(** AXIS Z **)
	(* Brake timer *)
		tonZBrake(PT:=T#20S);
		IF GV_Axes.stAxisZ.bPowerEnable AND GV_Axes.stAxisZ.stDriveAx8206.AxisRef.Status.NotMoving THEN
			tonZBrake.IN:=TRUE;
		ELSE
			tonZBrake.IN:=FALSE;
		END_IF
	(* Setup *)
		GV_Axes.stAxisZ.bPresence:=TRUE; // Axis Presence
		fbEventGroupAssignement(iEventGroup:=GV_Axes.stAxisZ.iEventGroup);
		GV_Axes.stAxisZ.strIdHMI:='Z'; // String for events on HMI
		GV_Axes.stAxisZ.iIdHMI:=UDINT_TO_INT(GV_Axes.stAxisZ.stDriveAx8206.AxisRef.NcToPlc.AxisId); // Number for events on HMI
		(*Power*)
			IF ((GV_OpMode.eOpMode=ENUM_OpMode.INIT AND (GV_Axes.stAxisZ.bAutoCmdAbs OR (GV_Axes.stAxisZ.bPowerEnable AND (NOT tonZBrake.Q)))) // INIT
			OR (GV_OpMode.eOpMode=ENUM_OpMode.AUTO AND (GV_Axes.stAxisZ.bAutoCmdAbs OR (GV_Axes.stAxisZ.bPowerEnable AND (NOT tonZBrake.Q)))) // AUTO
			OR (GV_OpMode.eOpMode=ENUM_OpMode.MANU AND (((NOT GV_Handwheel.aId[1].bEnable) AND (GV_Axes.eJogAxisRequest=ENUM_Axis_Select.Z OR GV_Axes.eJogAxisSelect=ENUM_Axis_Select.Z)) OR (GV_Handwheel.aId[1].bEnable AND GV_Handwheel.aId[1].eAxisSelect=ENUM_Axis_Select.Z)))) // MANU
			AND ((GV_General.bSafety AND GV_General.bPower AND (NOT GV_Axes.stAxisZ.bAlAxisFault)) OR (GV_Axes.stAxisZ.bPowerEnable AND ((GV_Axes.stAxisZ.bStopExecute AND (NOT GV_Axes.stAxisZ.bStopDone))) OR (GV_Axes.stAxisZ.bHaltExecute AND (NOT GV_Axes.stAxisZ.bHaltDone)))) AND (NOT GV_General.bRebootRequest) AND (NOT GV_General.bShutdownRequest) THEN
				GV_Axes.stAxisZ.bPowerEnable:=TRUE;
			ELSE
				GV_Axes.stAxisZ.bPowerEnable:=FALSE;
			END_IF
		(*Stop*)
			GV_Axes.stAxisZ.bStopExecute:=(NOT GV_General.bSafety) OR (NOT GV_General.bPower) OR GV_General.bRebootRequest OR GV_General.bShutdownRequest (*OR (GV_OpMode.eOpMode=ENUM_OpMode.AUTO AND GV_Cycle.bCycleInProgress AND (NOT GV_Cycle.bStartStop))*); // Have to stop
		(*Halt*)
			GV_Axes.stAxisZ.bHaltExecute:=(GV_OpMode.eOpMode=ENUM_OpMode.AUTO AND GV_Cycle.bCycleInProgress AND (NOT GV_Cycle.bStartStop)); // Have to halt
		(*Abort*)
			//GV_Axes.stAxisZ.bAbort:=(NOT GV_Axes.stAxisZ.stDriveAx8206.AxisRef.Status.NotMoving) AND (GV_OpMode.eOpMode=ENUM_OpMode.AUTO AND GV_Cycle.bCycleInProgress AND (NOT GV_Cycle.bStartStop)); // Have to abort
		(*Reset*)
			GV_Axes.stAxisZ.bEventAck:=GV_HMI.bEventAck; // Events Acknowledgement	
		(*Jog*)
			GV_Axes.stAxisZ.bJogEnable:=GV_OpMode.eOpMode=ENUM_OpMode.MANU AND GV_Axes.stAxisZ.stDriveAx8206.AxisRef.Status.Operational AND (NOT GV_Axes.stAxisZ.bAlAxisFault) AND
			((GV_Handwheel.aId[1].bEnable AND GV_Handwheel.aId[1].eAxisSelect=ENUM_Axis_Select.Z) OR ((NOT GV_Handwheel.aId[1].bEnable) AND GV_HMI.iCurrentScreenNumber=210 AND GV_Axes.eJogAxisSelect=ENUM_Axis_Select.Z));
			IF GV_Axes.stAxisZ.bJogEnable AND (NOT GV_Handwheel.aId[1].bEnable) THEN // Jog from HMI
				GV_Axes.stAxisZ.eJogMode:=TC2_MC2.E_JogMode.MC_JOGMODE_CONTINOUS; // Jog Mode
				GV_Axes.stAxisZ.bJogPlus:=GV_HMI.stAxes.bButtonPlus; // Jog +
				GV_Axes.stAxisZ.bJogMinus:=GV_HMI.stAxes.bButtonMinus; // Jog -
				GV_Axes.stAxisZ.lrJogPos:=0; // Jog Position -> Only in mode INCHING
				GV_Axes.stAxisZ.lrJogVel:=GV_Axes.lrVelocityAxisZ; // Jog Velocity
				GV_Axes.stAxisZ.lrJogAcc:=0; // Jog Acceleration -> see the Axis Configuration in the System Manager
				GV_Axes.stAxisZ.lrJogDec:=0; // Jog Decelration -> see the Axis Configuration in the System Manager
				GV_Axes.stAxisZ.lrJogJerk:=0; // Jog Jerk -> see the Axis Configuration in the System Manager
			ELSIF GV_Axes.stAxisZ.bJogEnable AND GV_Handwheel.aId[1].bEnable AND GV_Handwheel.aId[1].bJogRequestRisingEdge THEN // Jog from Handwheel
				GV_Axes.stAxisZ.eJogMode:=TC2_MC2.E_JogMode.MC_JOGMODE_INCHING; // Jog Mode
				GV_Axes.stAxisZ.bJogPlus:=(GV_Handwheel.aId[1].eJogDirection=ENUM_Jog_Direction.Plus); // Jog +
				GV_Axes.stAxisZ.bJogMinus:=(GV_Handwheel.aId[1].eJogDirection=ENUM_Jog_Direction.Minus); // Jog -
				GV_Axes.stAxisZ.lrJogPos:=GV_Handwheel.aId[1].lrJogIncrRequest; // Jog Position
				GV_Axes.stAxisZ.lrJogVel:=GV_Axes.lrJogMaxSpeedAxisZ;//GV_Axes.lrVelocityAxisZ; // Jog Velocity
				GV_Axes.stAxisZ.lrJogAcc:=0; // Jog Acceleration -> see the Axis Configuration in the System Manager
				GV_Axes.stAxisZ.lrJogDec:=0; // Jog Decelration -> see the Axis Configuration in the System Manager
				GV_Axes.stAxisZ.lrJogJerk:=0; // Jog Jerk -> see the Axis Configuration in the System Manager
			ELSE
				GV_Axes.stAxisZ.bJogPlus:=FALSE; // Jog +
				GV_Axes.stAxisZ.bJogMinus:=FALSE; // Jog -
				GV_Axes.stAxisZ.lrJogPos:=0; // Jog Position
				GV_Axes.stAxisZ.lrJogVel:=0; // Jog Velocity
				GV_Axes.stAxisZ.lrJogAcc:=0; // Jog Acceleration -> see the Axis Configuration in the System Manager
				GV_Axes.stAxisZ.lrJogDec:=0; // Jog Decelration -> see the Axis Configuration in the System Manager
				GV_Axes.stAxisZ.lrJogJerk:=0; // Jog Jerk -> see the Axis Configuration in the System Manager				
			END_IF
		(*AUTO*)
			GV_Axes.stAxisZ.bAutoEnable:=GV_OpMode.eOpMode=ENUM_OpMode.AUTO AND GV_Cycle.bStartStop AND GV_Axes.stAxisZ.stDriveAx8206.AxisRef.Status.Operational AND (NOT GV_Axes.stAxisZ.bAlAxisFault);
			IF  GV_Axes.stAxisZ.bAutoEnable THEN
				GV_Axes.stAxisZ.lrAutoVelAbs:=GV_Axes.lrVelocityAxisZ; // AUTO Velocity
				GV_Axes.stAxisZ.lrAutoAccAbs:=0; // AUTO Acceleration -> see the Axis Configuration in the System Manager
				GV_Axes.stAxisZ.lrAutoDecAbs:=0; // AUTO Decelration -> see the Axis Configuration in the System Manager
				GV_Axes.stAxisZ.lrAutoJerkAbs:=0; // AUTO Jerk -> see the Axis Configuration in the System Manager
			ELSE
				GV_Axes.stAxisZ.lrAutoVelAbs:=0; // AUTO Velocity
				GV_Axes.stAxisZ.lrAutoAccAbs:=0; // AUTO Acceleration -> see the Axis Configuration in the System Manager
				GV_Axes.stAxisZ.lrAutoDecAbs:=0; // AUTO Decelration -> see the Axis Configuration in the System Manager
				GV_Axes.stAxisZ.lrAutoJerkAbs:=0; // AUTO Jerk -> see the Axis Configuration in the System Manager
			END_IF
		(*Referencing*)
			GV_Axes.stAxisZ.bSetOffsetExecute:=GV_OpMode.eOpMode=ENUM_OpMode.MANU AND GV_Axes.stAxisZ.stDriveAx8206.AxisRef.Status.Operational AND (NOT GV_Axes.stAxisZ.bAlAxisFault) AND GV_HMI.iCurrentScreenNumber=308 AND GV_Axes.eRefAxisSelect=ENUM_Axis_Select.Z AND GV_HMI.stAxes.rtButtonReferencingAxis.Q;
			GV_Axes.stAxisZ.bDeleteOffsetExecute:=FALSE; // Not used in the HMI, we can use it from here or add it in the HMI later if it's necessary	
		(*ReadParameter BOOL*)
			GV_Axes.stAxisZ.bReadbEnable:=(GV_Axes.stAxisZ.mcAxisReadParameterb=MC_AxisParameter.AxisEnMinSoftPosLimit OR GV_Axes.stAxisZ.mcAxisReadParameterb=MC_AxisParameter.AxisEnMaxSoftPosLimit) AND GV_Axes.stAxisZ.stDriveAx8206.AxisRef.Status.Operational;
			IF GV_Axes.stAxisZ.stDriveAx8206.AxisRef.Status.Operational THEN
				IF GV_Axes.stAxisZ.mcAxisReadParameterb=MC_AxisParameter.AxisEnMaxSoftPosLimit THEN
					IF GV_General.bIsBlinking05s THEN
						GV_Axes.stAxisZ.mcAxisReadParameterb:=MC_AxisParameter.AxisEnMinSoftPosLimit;
					ELSE
						IF GV_Axes.stAxisZ.bReadbValid THEN
							GV_Axes.stAxisZ.bReadEnMaxSoftPosLimit:=GV_Axes.stAxisZ.bReadbValue;
						END_IF
					END_IF
				ELSIF GV_Axes.stAxisZ.mcAxisReadParameterb=MC_AxisParameter.AxisEnMinSoftPosLimit THEN
					IF GV_General.bIsBlinking05s THEN
						GV_Axes.stAxisZ.mcAxisReadParameterb:=MC_AxisParameter.AxisEnMaxSoftPosLimit;
					ELSE
						IF GV_Axes.stAxisZ.bReadbValid THEN
							GV_Axes.stAxisZ.bReadEnMinSoftPosLimit:=GV_Axes.stAxisZ.bReadbValue;
						END_IF
					END_IF
				ELSE
					GV_Axes.stAxisZ.mcAxisReadParameterb:=MC_AxisParameter.AxisEnMinSoftPosLimit;
				END_IF
			END_IF
		(*ReadParameter LREAL*)
			GV_Axes.stAxisZ.bReadlrEnable:=(GV_Axes.stAxisZ.mcAxisReadParameterlr=MC_AxisParameter.AxisMinSoftPosLimit OR GV_Axes.stAxisZ.mcAxisReadParameterlr=MC_AxisParameter.AxisMaxSoftPosLimit) AND GV_Axes.stAxisZ.stDriveAx8206.AxisRef.Status.Operational;
			IF GV_Axes.stAxisZ.stDriveAx8206.AxisRef.Status.Operational THEN
				IF GV_Axes.stAxisZ.mcAxisReadParameterlr=MC_AxisParameter.AxisMaxSoftPosLimit THEN
					IF GV_General.bIsBlinking05s THEN
						GV_Axes.stAxisZ.mcAxisReadParameterlr:=MC_AxisParameter.AxisMinSoftPosLimit;
					ELSE
						IF GV_Axes.stAxisZ.bReadlrValid THEN
							GV_Axes.stAxisZ.lrReadMaxSoftPosLimit:=GV_Axes.stAxisZ.lrReadlrValue;
						END_IF
					END_IF
				ELSIF GV_Axes.stAxisZ.mcAxisReadParameterlr=MC_AxisParameter.AxisMinSoftPosLimit THEN
					IF (NOT GV_General.bIsBlinking05s) THEN
						GV_Axes.stAxisZ.mcAxisReadParameterlr:=MC_AxisParameter.AxisMaxSoftPosLimit;
					ELSE
						IF GV_Axes.stAxisZ.bReadlrValid THEN
							GV_Axes.stAxisZ.lrReadMinSoftPosLimit:=GV_Axes.stAxisZ.lrReadlrValue;
						END_IF
					END_IF
				ELSE
					GV_Axes.stAxisZ.mcAxisReadParameterlr:=MC_AxisParameter.AxisMinSoftPosLimit;
				END_IF
			END_IF	
		(*WriteParameter BOOL*)
// 			GV_Axes.stAxisZ.bWritebExecute:=GV_Axes.eRefAxisSelect=ENUM_Axis_Select.Z AND (GV_HMI.stAxes.rtButtonMinSofltLimit.Q OR GV_HMI.stAxes.rtButtonMaxSofltLimit.Q) AND GV_Axes.stAxisZ.stDriveAx8206.AxisRef.Status.Operational;
// 			IF GV_Axes.stAxisZ.stDriveAx8206.AxisRef.Status.Operational AND (NOT GV_Axes.stAxisZ.stDriveAx8206.AxisRef.Status.Moving) THEN
// 				IF GV_HMI.stAxes.rtButtonMinSofltLimit.Q THEN
// 					GV_Axes.stAxisZ.mcAxisWriteParameterb:=MC_AxisParameter.AxisEnMinSoftPosLimit;
// 					IF GV_Axes.stAxisZ.bReadEnMinSoftPosLimit THEN
// 						GV_Axes.stAxisZ.bWritebValue:=FALSE;
// 					ELSE
// 						GV_Axes.stAxisZ.bWritebValue:=TRUE;
// 					END_IF
// 				ELSIF GV_HMI.stAxes.rtButtonMaxSofltLimit.Q THEN
// 					GV_Axes.stAxisZ.mcAxisWriteParameterb:=MC_AxisParameter.AxisEnMaxSoftPosLimit;
// 					IF GV_Axes.stAxisZ.bReadEnMaxSoftPosLimit THEN
// 						GV_Axes.stAxisZ.bWritebValue:=FALSE;
// 					ELSE
// 						GV_Axes.stAxisZ.bWritebValue:=TRUE;
// 					END_IF
// 				END_IF
// 			END_IF
		(*WriteParameter LREAL*)
// 			bAxisZWrite1:=FALSE;
// 			bAxisZWrite2:=FALSE;
// 			bAxisZWrite3:=FALSE;
// 			bAxisZWrite4:=FALSE;
// 			IF GV_Tool_Magazine.stManipulator.ePositionMag=ENUM_Position_Magazine.Top THEN
// 				IF GV_Tool_Magazine.stManipulator.lrZPosition<>GV_Tool_Magazine.stManipulator.lrZTunnel THEN
// 					GV_Axes.stAxisZ.lrValueMax:=-10;
// 					GV_Axes.stAxisZ.lrValueMin:=-350;
// 					bAxisZWrite1:=TRUE;
// 				ELSE
// 					GV_Axes.stAxisZ.lrValueMax:=-10;
// 					GV_Axes.stAxisZ.lrValueMin:=-800;
// 					bAxisZWrite2:=TRUE;
// 				END_IF
// 			END_IF
// 			IF GV_Tool_Magazine.stManipulator.ePositionMag=ENUM_Position_Magazine.Bottom THEN
// 				IF GV_Tool_Magazine.stManipulator.lrZPosition<>GV_Tool_Magazine.stManipulator.lrZTunnel THEN
// 					GV_Axes.stAxisZ.lrValueMax:=-450;
// 					GV_Axes.stAxisZ.lrValueMin:=-800;
// 					bAxisZWrite3:=TRUE;
// 				ELSE
// 					GV_Axes.stAxisZ.lrValueMax:=-10;
// 					GV_Axes.stAxisZ.lrValueMin:=-800;
// 					bAxisZWrite4:=TRUE;
// 				END_IF
// 			END_IF
// 			rtAxisZWrite1(CLK:=bAxisZWrite1);
// 			rtAxisZWrite2(CLK:=bAxisZWrite2);
// 			rtAxisZWrite3(CLK:=bAxisZWrite3);
// 			rtAxisZWrite4(CLK:=bAxisZWrite4);
// 			IF rtAxisZWrite1.Q OR rtAxisZWrite2.Q OR rtAxisZWrite3.Q OR rtAxisZWrite4.Q THEN
// 				GV_Axes.stAxisZ.mcAxisWriteParameterlr:=MC_AxisParameter.AxisMaxSoftPosLimit;
// 				GV_Axes.stAxisZ.lrWritelrValue:=GV_Axes.stAxisZ.lrValueMax;
// 				bAxisZWriteMin:=FALSE;
// 				bAxisZWriteMax:=TRUE;
// 			END_IF
// 			IF bAxisZWriteMax AND GV_Axes.stAxisZ.bWritelrBusy THEN
// 				GV_Axes.stAxisZ.mcAxisWriteParameterlr:=MC_AxisParameter.AxisMinSoftPosLimit;
// 				GV_Axes.stAxisZ.lrWritelrValue:=GV_Axes.stAxisZ.lrValueMin;
// 				bAxisZWriteMin:=TRUE;
// 				bAxisZWriteMax:=FALSE;
// 			END_IF
// 			IF bAxisZWriteMin AND GV_Axes.stAxisZ.bWritelrBusy THEN
// 				bAxisZWriteMin:=FALSE;
// 				bAxisZWriteMax:=FALSE;
// 			END_IF
// 			GV_Axes.stAxisZ.bWritelrExecute:=(bAxisZWriteMax OR bAxisZWriteMin) AND GV_Axes.stAxisZ.bWritelrDone AND (NOT GV_Axes.stAxisZ.bWritelrBusy) AND GV_Axes.stAxisZ.stDriveAx8206.AxisRef.Status.Operational;
// 			
	(* Fb *)
		IF GV_Axes.stAxisZ.bPresence THEN
			fbAxisZ(
					stAxis:=GV_Axes.stAxisZ,
					);
		END_IF

(** AXIS Arm **)
	(* Setup *)
		GV_Axes.stAxisArm.bPresence:=TRUE; // Axis Presence
		fbEventGroupAssignement(iEventGroup:=GV_Axes.stAxisArm.iEventGroup);
		GV_Axes.stAxisArm.strIdHMI:='Arm'; // String for events on HMI
		GV_Axes.stAxisArm.iIdHMI:=UDINT_TO_INT(GV_Axes.stAxisArm.stDriveAx8206.AxisRef.NcToPlc.AxisId); // Number for events on HMI
		(*Power*)
			IF ((GV_General.bSafety AND GV_General.bPower AND (NOT GV_Axes.stAxisArm.bAlAxisFault)) OR (GV_Axes.stAxisArm.bPowerEnable AND ((GV_Axes.stAxisArm.bStopExecute AND (NOT GV_Axes.stAxisArm.bStopDone))) OR ((GV_Axes.stAxisArm.bHaltExecute AND (NOT GV_Axes.stAxisArm.bHaltDone))))) AND (NOT GV_General.bRebootRequest) AND (NOT GV_General.bShutdownRequest) THEN
				GV_Axes.stAxisArm.bPowerEnable:=TRUE;
			ELSE
				GV_Axes.stAxisArm.bPowerEnable:=FALSE;
			END_IF
		(*Stop*)
			GV_Axes.stAxisArm.bStopExecute:=(NOT GV_General.bSafety) OR (NOT GV_General.bPower) OR GV_General.bRebootRequest OR GV_General.bShutdownRequest (*OR (GV_OpMode.eOpMode=ENUM_OpMode.AUTO AND GV_Cycle.bCycleInProgress AND (NOT GV_Cycle.bStartStop))*); // Have to stop
		(*Halt*)
			GV_Axes.stAxisArm.bHaltExecute:=(GV_OpMode.eOpMode=ENUM_OpMode.AUTO AND GV_Cycle.bCycleInProgress AND (NOT GV_Cycle.bStartStop)); // Have to halt
		(*Abort*)
			//GV_Axes.stAxisArm.bAbort:=(NOT GV_Axes.stAxisArm.stDriveAx8206.AxisRef.Status.NotMoving) AND (GV_OpMode.eOpMode=ENUM_OpMode.AUTO AND GV_Cycle.bCycleInProgress AND (NOT GV_Cycle.bStartStop)); // Have to abort
		(*Reset*)
			GV_Axes.stAxisArm.bEventAck:=GV_HMI.bEventAck; // Events Acknowledgement	
		(*Jog*)
			GV_Axes.stAxisArm.bJogEnable:=GV_OpMode.eOpMode=ENUM_OpMode.MANU AND GV_Axes.stAxisArm.stDriveAx8206.AxisRef.Status.Operational AND (NOT GV_Axes.stAxisArm.bAlAxisFault) AND
			((GV_Handwheel.aId[1].bEnable AND GV_Handwheel.aId[1].eAxisSelect=ENUM_Axis_Select.Arm) OR ((NOT GV_Handwheel.aId[1].bEnable) AND GV_HMI.iCurrentScreenNumber=210 AND GV_Axes.eJogAxisSelect=ENUM_Axis_Select.Arm));
			IF GV_Axes.stAxisArm.bJogEnable AND (NOT GV_Handwheel.aId[1].bEnable) THEN // Jog from HMI
				GV_Axes.stAxisArm.eJogMode:=TC2_MC2.E_JogMode.MC_JOGMODE_CONTINOUS; // Jog Mode
				GV_Axes.stAxisArm.bJogPlus:=GV_HMI.stAxes.bButtonPlus; // Jog +
				GV_Axes.stAxisArm.bJogMinus:=GV_HMI.stAxes.bButtonMinus; // Jog -
				GV_Axes.stAxisArm.lrJogPos:=0; // Jog Position -> Only in mode INCHING
				GV_Axes.stAxisArm.lrJogVel:=GV_Axes.lrVelocityAxisArm; // Jog Velocity
				GV_Axes.stAxisArm.lrJogAcc:=0; // Jog Acceleration -> see the Axis Configuration in the System Manager
				GV_Axes.stAxisArm.lrJogDec:=0; // Jog Decelration -> see the Axis Configuration in the System Manager
				GV_Axes.stAxisArm.lrJogJerk:=0; // Jog Jerk -> see the Axis Configuration in the System Manager
			ELSIF GV_Axes.stAxisArm.bJogEnable AND GV_Handwheel.aId[1].bEnable AND GV_Handwheel.aId[1].bJogRequestRisingEdge THEN // Jog from Handwheel
				GV_Axes.stAxisArm.eJogMode:=TC2_MC2.E_JogMode.MC_JOGMODE_INCHING; // Jog Mode
				GV_Axes.stAxisArm.bJogPlus:=(GV_Handwheel.aId[1].eJogDirection=ENUM_Jog_Direction.Plus); // Jog +
				GV_Axes.stAxisArm.bJogMinus:=(GV_Handwheel.aId[1].eJogDirection=ENUM_Jog_Direction.Minus); // Jog -
				GV_Axes.stAxisArm.lrJogPos:=GV_Handwheel.aId[1].lrJogIncrRequest; // Jog Position
				GV_Axes.stAxisArm.lrJogVel:=GV_Axes.lrJogMaxSpeedAxisArm;//GV_Axes.lrVelocityAxisArm; // Jog Velocity
				GV_Axes.stAxisArm.lrJogAcc:=0; // Jog Acceleration -> see the Axis Configuration in the System Manager
				GV_Axes.stAxisArm.lrJogDec:=0; // Jog Decelration -> see the Axis Configuration in the System Manager
				GV_Axes.stAxisArm.lrJogJerk:=0; // Jog Jerk -> see the Axis Configuration in the System Manager
			ELSE
				GV_Axes.stAxisArm.bJogPlus:=FALSE; // Jog +
				GV_Axes.stAxisArm.bJogMinus:=FALSE; // Jog -
				GV_Axes.stAxisArm.lrJogPos:=0; // Jog Position
				GV_Axes.stAxisArm.lrJogVel:=0; // Jog Velocity
				GV_Axes.stAxisArm.lrJogAcc:=0; // Jog Acceleration -> see the Axis Configuration in the System Manager
				GV_Axes.stAxisArm.lrJogDec:=0; // Jog Decelration -> see the Axis Configuration in the System Manager
				GV_Axes.stAxisArm.lrJogJerk:=0; // Jog Jerk -> see the Axis Configuration in the System Manager				
			END_IF
		(*AUTO*)
			GV_Axes.stAxisArm.bAutoEnable:=GV_OpMode.eOpMode=ENUM_OpMode.AUTO AND GV_Cycle.bStartStop AND GV_Axes.stAxisArm.stDriveAx8206.AxisRef.Status.Operational AND (NOT GV_Axes.stAxisArm.bAlAxisFault);
			IF  GV_Axes.stAxisArm.bAutoEnable THEN
				GV_Axes.stAxisArm.lrAutoVelAbs:=GV_Axes.lrVelocityAxisArm; // AUTO Velocity
				GV_Axes.stAxisArm.lrAutoAccAbs:=0; // AUTO Acceleration -> see the Axis Configuration in the System Manager
				GV_Axes.stAxisArm.lrAutoDecAbs:=0; // AUTO Decelration -> see the Axis Configuration in the System Manager
				GV_Axes.stAxisArm.lrAutoJerkAbs:=0; // AUTO Jerk -> see the Axis Configuration in the System Manager
			ELSE
				GV_Axes.stAxisArm.lrAutoVelAbs:=0; // AUTO Velocity
				GV_Axes.stAxisArm.lrAutoAccAbs:=0; // AUTO Acceleration -> see the Axis Configuration in the System Manager
				GV_Axes.stAxisArm.lrAutoDecAbs:=0; // AUTO Decelration -> see the Axis Configuration in the System Manager
				GV_Axes.stAxisArm.lrAutoJerkAbs:=0; // AUTO Jerk -> see the Axis Configuration in the System Manager
			END_IF
		(*Referencing*)
			GV_Axes.stAxisArm.bSetOffsetExecute:=GV_OpMode.eOpMode=ENUM_OpMode.MANU AND GV_Axes.stAxisArm.stDriveAx8206.AxisRef.Status.Operational AND (NOT GV_Axes.stAxisArm.bAlAxisFault) AND GV_HMI.iCurrentScreenNumber=308 AND GV_Axes.eRefAxisSelect=ENUM_Axis_Select.Arm AND GV_HMI.stAxes.rtButtonReferencingAxis.Q;
			GV_Axes.stAxisArm.bDeleteOffsetExecute:=FALSE; // Not used in the HMI, we can use it from here or add it in the HMI later if it's necessary	
		(*ReadParameter BOOL*)
			GV_Axes.stAxisArm.bReadbEnable:=(GV_Axes.stAxisArm.mcAxisReadParameterb=MC_AxisParameter.AxisEnMinSoftPosLimit OR GV_Axes.stAxisArm.mcAxisReadParameterb=MC_AxisParameter.AxisEnMaxSoftPosLimit) AND GV_Axes.stAxisArm.stDriveAx8206.AxisRef.Status.Operational;
			IF GV_Axes.stAxisArm.stDriveAx8206.AxisRef.Status.Operational THEN
				IF GV_Axes.stAxisArm.mcAxisReadParameterb=MC_AxisParameter.AxisEnMaxSoftPosLimit THEN
					IF GV_General.bIsBlinking05s THEN
						GV_Axes.stAxisArm.mcAxisReadParameterb:=MC_AxisParameter.AxisEnMinSoftPosLimit;
					ELSE
						IF GV_Axes.stAxisArm.bReadbValid THEN
							GV_Axes.stAxisArm.bReadEnMaxSoftPosLimit:=GV_Axes.stAxisArm.bReadbValue;
						END_IF
					END_IF
				ELSIF GV_Axes.stAxisArm.mcAxisReadParameterb=MC_AxisParameter.AxisEnMinSoftPosLimit THEN
					IF GV_General.bIsBlinking05s THEN
						GV_Axes.stAxisArm.mcAxisReadParameterb:=MC_AxisParameter.AxisEnMaxSoftPosLimit;
					ELSE
						IF GV_Axes.stAxisArm.bReadbValid THEN
							GV_Axes.stAxisArm.bReadEnMinSoftPosLimit:=GV_Axes.stAxisArm.bReadbValue;
						END_IF
					END_IF
				ELSE
					GV_Axes.stAxisArm.mcAxisReadParameterb:=MC_AxisParameter.AxisEnMinSoftPosLimit;
				END_IF
			END_IF
		(*ReadParameter LREAL*)
			GV_Axes.stAxisArm.bReadlrEnable:=(GV_Axes.stAxisArm.mcAxisReadParameterlr=MC_AxisParameter.AxisMinSoftPosLimit OR GV_Axes.stAxisArm.mcAxisReadParameterlr=MC_AxisParameter.AxisMaxSoftPosLimit) AND GV_Axes.stAxisArm.stDriveAx8206.AxisRef.Status.Operational;
			IF GV_Axes.stAxisArm.stDriveAx8206.AxisRef.Status.Operational THEN
				IF GV_Axes.stAxisArm.mcAxisReadParameterlr=MC_AxisParameter.AxisMaxSoftPosLimit THEN
					IF GV_General.bIsBlinking05s THEN
						GV_Axes.stAxisArm.mcAxisReadParameterlr:=MC_AxisParameter.AxisMinSoftPosLimit;
					ELSE
						IF GV_Axes.stAxisArm.bReadlrValid THEN
							GV_Axes.stAxisArm.lrReadMaxSoftPosLimit:=GV_Axes.stAxisArm.lrReadlrValue;
						END_IF
					END_IF
				ELSIF GV_Axes.stAxisArm.mcAxisReadParameterlr=MC_AxisParameter.AxisMinSoftPosLimit THEN
					IF (NOT GV_General.bIsBlinking05s) THEN
						GV_Axes.stAxisArm.mcAxisReadParameterlr:=MC_AxisParameter.AxisMaxSoftPosLimit;
					ELSE
						IF GV_Axes.stAxisArm.bReadlrValid THEN
							GV_Axes.stAxisArm.lrReadMinSoftPosLimit:=GV_Axes.stAxisArm.lrReadlrValue;
						END_IF
					END_IF
				ELSE
					GV_Axes.stAxisArm.mcAxisReadParameterlr:=MC_AxisParameter.AxisMinSoftPosLimit;
				END_IF
			END_IF	
		(*WriteParameter BOOL*)
// 			GV_Axes.stAxisArm.bWritebExecute:=GV_Axes.eRefAxisSelect=ENUM_Axis_Select.Arm AND (GV_HMI.stAxes.rtButtonMinSofltLimit.Q OR GV_HMI.stAxes.rtButtonMaxSofltLimit.Q) AND GV_Axes.stAxisArm.stDriveAx8206.AxisRef.Status.Operational;
// 			IF GV_Axes.stAxisArm.stDriveAx8206.AxisRef.Status.Operational AND (NOT GV_Axes.stAxisArm.stDriveAx8206.AxisRef.Status.Moving) THEN
// 				IF GV_HMI.stAxes.rtButtonMinSofltLimit.Q THEN
// 					GV_Axes.stAxisArm.mcAxisWriteParameterb:=MC_AxisParameter.AxisEnMinSoftPosLimit;
// 					IF GV_Axes.stAxisArm.bReadEnMinSoftPosLimit THEN
// 						GV_Axes.stAxisArm.bWritebValue:=FALSE;
// 					ELSE
// 						GV_Axes.stAxisArm.bWritebValue:=TRUE;
// 					END_IF
// 				ELSIF GV_HMI.stAxes.rtButtonMaxSofltLimit.Q THEN
// 					GV_Axes.stAxisArm.mcAxisWriteParameterb:=MC_AxisParameter.AxisEnMaxSoftPosLimit;
// 					IF GV_Axes.stAxisArm.bReadEnMaxSoftPosLimit THEN
// 						GV_Axes.stAxisArm.bWritebValue:=FALSE;
// 					ELSE
// 						GV_Axes.stAxisArm.bWritebValue:=TRUE;
// 					END_IF
// 				END_IF
// 			END_IF
		(*WriteParameter LREAL*)
// 			bAxisArmWrite1:=FALSE;
// 			bAxisArmWrite2:=FALSE;
// 			bAxisArmWrite3:=FALSE;
// 			bAxisArmWrite4:=FALSE;
// 			IF GV_Tool_Magazine.stManipulator.ePositionMag=ENUM_Position_Magazine.Top THEN
// 				IF GV_Tool_Magazine.stManipulator.lrArmPosition<>GV_Tool_Magazine.stManipulator.lrArmTunnel THEN
// 					GV_Axes.stAxisArm.lrValueMax:=-10;
// 					GV_Axes.stAxisArm.lrValueMin:=-350;
// 					bAxisArmWrite1:=TRUE;
// 				ELSE
// 					GV_Axes.stAxisArm.lrValueMax:=-10;
// 					GV_Axes.stAxisArm.lrValueMin:=-800;
// 					bAxisArmWrite2:=TRUE;
// 				END_IF
// 			END_IF
// 			IF GV_Tool_Magazine.stManipulator.ePositionMag=ENUM_Position_Magazine.Bottom THEN
// 				IF GV_Tool_Magazine.stManipulator.lrArmPosition<>GV_Tool_Magazine.stManipulator.lrArmTunnel THEN
// 					GV_Axes.stAxisArm.lrValueMax:=-450;
// 					GV_Axes.stAxisArm.lrValueMin:=-800;
// 					bAxisArmWrite3:=TRUE;
// 				ELSE
// 					GV_Axes.stAxisArm.lrValueMax:=-10;
// 					GV_Axes.stAxisArm.lrValueMin:=-800;
// 					bAxisArmWrite4:=TRUE;
// 				END_IF
// 			END_IF
// 			rtAxisArmWrite1(CLK:=bAxisArmWrite1);
// 			rtAxisArmWrite2(CLK:=bAxisArmWrite2);
// 			rtAxisArmWrite3(CLK:=bAxisArmWrite3);
// 			rtAxisArmWrite4(CLK:=bAxisArmWrite4);
// 			IF rtAxisArmWrite1.Q OR rtAxisArmWrite2.Q OR rtAxisArmWrite3.Q OR rtAxisArmWrite4.Q THEN
// 				GV_Axes.stAxisArm.mcAxisWriteParameterlr:=MC_AxisParameter.AxisMaxSoftPosLimit;
// 				GV_Axes.stAxisArm.lrWritelrValue:=GV_Axes.stAxisArm.lrValueMax;
// 				bAxisArmWriteMin:=FALSE;
// 				bAxisArmWriteMax:=TRUE;
// 			END_IF
// 			IF bAxisArmWriteMax AND GV_Axes.stAxisArm.bWritelrBusy THEN
// 				GV_Axes.stAxisArm.mcAxisWriteParameterlr:=MC_AxisParameter.AxisMinSoftPosLimit;
// 				GV_Axes.stAxisArm.lrWritelrValue:=GV_Axes.stAxisArm.lrValueMin;
// 				bAxisArmWriteMin:=TRUE;
// 				bAxisArmWriteMax:=FALSE;
// 			END_IF
// 			IF bAxisArmWriteMin AND GV_Axes.stAxisArm.bWritelrBusy THEN
// 				bAxisArmWriteMin:=FALSE;
// 				bAxisArmWriteMax:=FALSE;
// 			END_IF
// 			GV_Axes.stAxisArm.bWritelrExecute:=(bAxisArmWriteMax OR bAxisArmWriteMin) AND GV_Axes.stAxisArm.bWritelrDone AND (NOT GV_Axes.stAxisArm.bWritelrBusy) AND GV_Axes.stAxisArm.stDriveAx8206.AxisRef.Status.Operational;
// 			
	(* Fb *)
		IF GV_Axes.stAxisArm.bPresence THEN
			fbAxisArm(
					stAxis:=GV_Axes.stAxisArm,
					);
		END_IF

(* Axis Disabled *)
	GV_Axes.bAxisAllDisabled:=GV_Axes.stAxisX.stDriveAx8206.AxisRef.Status.Disabled AND GV_Axes.stAxisY.stDriveAx8206.AxisRef.Status.Disabled AND GV_Axes.stAxisZ.stDriveAx8206.AxisRef.Status.Disabled AND GV_Axes.stAxisArm.stDriveAx8206.AxisRef.Status.Disabled;

(* Axis Not Moving *)
	GV_Axes.bAxisAllNotMoving:=GV_Axes.stAxisX.stDriveAx8206.AxisRef.Status.NotMoving AND GV_Axes.stAxisY.stDriveAx8206.AxisRef.Status.NotMoving AND GV_Axes.stAxisZ.stDriveAx8206.AxisRef.Status.NotMoving AND GV_Axes.stAxisArm.stDriveAx8206.AxisRef.Status.NotMoving;
	
(* Axis Operational *)
	GV_Axes.bAxisAllOperational:=GV_Axes.stAxisX.stDriveAx8206.AxisRef.Status.Operational AND GV_Axes.stAxisY.stDriveAx8206.AxisRef.Status.Operational AND GV_Axes.stAxisZ.stDriveAx8206.AxisRef.Status.Operational AND GV_Axes.stAxisArm.stDriveAx8206.AxisRef.Status.Operational;

END_PROGRAM

// ---- 10_Axes/03_POUs/02_FBs/FB_Axis.TcPOU
FUNCTION_BLOCK FB_Axis
VAR_INPUT	
END_VAR
VAR_OUTPUT
	(** PROCESS ENUM **)
	 	eStatus   : ENUM_Axis_Status ; // Status
END_VAR
VAR_IN_OUT
	(** AXIS_REF **)
		stAxis : ST_Axis ; // Axis structure
END_VAR	
VAR
	(** PROCESS LREAL **)
	
	(** PROCESS UDINT **)	
		(* mcPower *)
			udiPowerErrorId : UDINT ; // mcPower Error ID
		(* mcStop *)
			udiStopErrorId : UDINT ; // mcStop Error ID
		(* mcJog *)
			udiJogErrorId : UDINT ; // mcJog Error ID
		(* mcMoveAbs *)
			udiAutoErrorId : UDINT ; // mcMoveAbs Error ID
		(* mcReset *)
			udiResetErrorId : UDINT ; // mcReset Error ID
		(* mcReadbParameter*)
			udiReadbErrorId : UDINT ; // mcReadbParameter Error ID
		(* mcReadlrParameter*)
			udiReadlrErrorId : UDINT ; // mcReadlrParameter Error ID
		(* mcWritebParameter*)
			udiWritebErrorId : UDINT ; // mcWritebParameter Error ID
		(* mcWritelrParameter*)
			udiWritelrErrorId : UDINT ; // mcWritelrParameter Error ID
		(* fbSetPositionOffset*)
			udiSetPositionOffsetErrorId : UDINT ; // fbSetPositionOffset Error ID
		(* fbDeletePositionOffset*)
			udiDeletePositionOffsetErrorId : UDINT ; // fbDeletePositionOffset Error ID
			
	(** PROCESS FLAG **)
		bError : BOOL ; // Error
		bErrorParameter : BOOL ; // Error with mc parameter
		bErrorReferencing : BOOL ; // Error with fb referencing
		(* mcPower *)
			bPowered : BOOL ; // is Powered
			bPowerBusy : BOOL ; // mcPower Busy
			bPowerError : BOOL ; // mcPower Error
		(* mcStop *)
			bStopBusy : BOOL ; // mcStop Busy
			bStoping : BOOL ; // is Stoping
			bStopCmdAbort : BOOL ; // Stop Command Abort
			bStopError : BOOL ; // mcStop Error
		(* mcHalt *)
			bHaltBusy : BOOL ; // mcHalt Busy
			bHalting : BOOL ; // is Halting
			bHaltCmdAbort : BOOL ; // Halt Command Abort
			bHaltError : BOOL ; // mcHalt Error
		(* mcJog *)
			bJogBusy : BOOL ; // mcJog Busy
			bJogging : BOOL ; // is Moving in Jog
			bJogCmdAbort : BOOL ; // Jog Command Abort
			bJogError : BOOL ; // mcJog Error
		(* mcMoveAbs *)
			bAutoEnable : BOOL ; // Auto Enable
			//bAutoDone : BOOL ; // mcMoveAbs Done
			bAutoBusy : BOOL ; // mcMoveAbs Busy
			bAutoError : BOOL ; // mcMoveAbs Error
		(* mcReset *)
			bResetDone : BOOL ; // mcReset is Done
			bResetBusy : BOOL ; // mcReset is Busy
			bResetError : BOOL ; // mcReset Error
		(* mcReadbParameter*)
			bReadbBusy : BOOL ; // mcReadbParameter is Busy
			bReadbError : BOOL ; // mcReadbParameter Error
		(* mcReadlrParameter*)
			bReadlrBusy : BOOL ; // mcReadlPrarameter is Busy
			bReadlrError : BOOL ; // mcReadlrParameter Error
		(* mcWritebParameter*)
			//bWritebDone : BOOL ; // mcWritebParameter is Done
			//bWritebBusy : BOOL ; // mcWritebParameter is Busy
			bWritebError : BOOL ; // mcWritebParameter Error
		(* mcWritelrParameter*)
			//bWritelrDone : BOOL ; // mcWritelrParameter is Done
			//bWritelrBusy : BOOL ; // mcWritelrParameter is Busy
			bWritelrError : BOOL ; // mcWritelrParameter Error
		(* fbSetPositionOffset *)
			bSetPositionOffsetBusy : BOOL ;  // fbSetPositionOffset is Busy
			bSetPositionOffsetError : BOOL ;  // fbSetPositionOffset Error
		(* fbDeletePositionOffset *)
			bDeletePositionOffsetBusy : BOOL ;  // fbDeletePositionOffset is Busy
			bDeletePositionOffsetError : BOOL ;  // fbDeletePositionOffset Error
			
	(** MC **)
		mcAxisPower: MC_Power ; // Bloc fonction, gère la mise sous puissance
		mcAxisStop : MC_Stop ; // Bloc fonction, gère le stop en cas de besoin
		mcAxisHalt : MC_Halt ; // Bloc fonction, gère le halt en cas de besoin
		mcAxisReset : MC_Reset ; // Bloc fonction, gère le reset 
		mcAxisJog : MC_Jog ; // Bloc fonction, déplacement manuel
		mcAxisMoveAbs : MC_MoveAbsolute ; // Bloc fonction, gère un déplacement absolue en position

		mcReadbParameter : MC_ReadBoolParameter ; // Bloc fondtion, lecture d'un parametre BOOL		
		mcReadlrParameter : MC_ReadParameter ; // Bloc fondtion, lecture d'un parametre LREAL
			//mcAxisReadParameter : MC_AxisParameter ; // Bloc fonction, choix paramètre de l'axe
		mcWritebParameter : MC_WriteBoolParameter ; // Bloc fondtion, écriture d'un parametre BOOL
		mcWritelrParameter : MC_WriteParameter ; // Bloc fondtion, écriture d'un parametre LREAL
			//mcAxisWriteParameter : MC_AxisParameter ; // Bloc fonction, choix paramètre de l'axe
		
	(** FB **)
		fbInitEvents : FB_Init_Events ;
		fbEventHMI : FB_Event_HMI ;
		
		fbSetPositionOffset : FB_CoEAX8000SetPositionOffset; // Bloc fonction, pour mise à 0 d'un Axe
		fbDeletePositionOffset : FB_CoEAX8000DeletePositionOffset; // Bloc fonction, pour enlever la mise à 0 d'un Axe
		
		tonPower : TON ; // Mise sous puissance retardé 
END_VAR

//-----------------------------------------------------------------------------------------
//
//                  					FB_Axis
//
//						Gestion générique d'un Axe avec codeur Absolu			
//-----------------------------------------------------------------------------------------
//
//Auteur: G.GOETZ
//Création: 29.01.2026
//Dernière modification : 29.01.2026 (G.GOETZ)
//       			
//-----------------------------------------------------------------------------------------
//
//     							Liste des modifications  	
//
// 29.01.2026 (G.GOETZ) -> Création		
//-----------------------------------------------------------------------------------------

// « FB_Axis est l’unique propriétaire de l’axe et gère tous les mouvements »

(** EVENTS **)
	IF GV_General.bFirstCycleTask OR GV_General.bFirstCycleSimu THEN
		GV_Events.aEventGroup[stAxis.iEventGroup].aAlarm[1].fbAlarm.CreateEx(TC_Events.AxisAlarms.Alarm1,TRUE,0);
		GV_Events.aEventGroup[stAxis.iEventGroup].aOpMessage[1].fbAlarm.CreateEx(TC_Events.AxisOpMessages.Message1,TRUE,0);	
		fbInitEvents(iEventGroup:=stAxis.iEventGroup,strEventType:='ALARM',strEventGuid:='40E67F82-65D4-40BA-B0A0-D5A8CC414B5C',tcEventSeverity:=2);
		fbInitEvents(iEventGroup:=stAxis.iEventGroup,strEventType:='OpMESSAGE',strEventGuid:='3D8607F0-0CB9-481C-A2EA-25B5E2E7FECD',tcEventSeverity:=1);
	END_IF	
		
(** ALARMS **)
	(* Axis fault *)
		(*Reset fault*)
			IF stAxis.bEventAck THEN
				stAxis.bAlAxisFault:=FALSE;
			END_IF
		(*Set fault*)
			IF stAxis.stDriveAx8206.AxisRef.NcToPlc.ErrorCode<>0 THEN
				stAxis.bAlAxisFault:=TRUE;
			END_IF
		(*Alarm 1 = Axis in fault*)
			IF stAxis.bAlAxisFault THEN
				GV_Events.aEventGroup[stAxis.iEventGroup].aAlarm[1].fbAlarm.ipArguments.Clear().AddString(stAxis.strIdHMI);
				fbEventHMI(iEventGroup:=stAxis.iEventGroup,iIdEvent:=1,strEventType:='ALARM',bEventSet:=TRUE);
			ELSE
				fbEventHMI(iEventGroup:=stAxis.iEventGroup,iIdEvent:=1,strEventType:='ALARM',bEventSet:=FALSE);			
			END_IF
			
(** MESSAGES **)




(** STATUS **)
	stAxis.stDriveAx8206.AxisRef.ReadStatus();

(** POWER **)
	(* tonPower *)
		tonPower(IN:=stAxis.bPowerEnable,PT:=T#250MS,Q=>,ET=>);
	(* mcPower *)
		mcAxisPower(
					// IN
					Axis:=stAxis.stDriveAx8206.AxisRef,
					Enable:=stAxis.bPowerEnable AND tonPower.Q,
					Enable_positive:=TRUE,
					Enable_negative:=TRUE,
					Override:=100, // = 100%
					BufferMode:=, // Not used
					Options:=, // Not used
					// OUT
					Status=>bPowered,
					Busy=>bPowerBusy,
					Error=>bPowerError,
					ErrorID=>udiPowerErrorId
					);

(** STOP **)
	(* mcStop *)
		mcAxisStop(
					//IN
					Axis:=stAxis.stDriveAx8206.AxisRef,
					Execute:=stAxis.bStopExecute,
					//Deceleration:=, // see the Axis Configuration in the System Manager
					//Jerk:=, // see the Axis Configuration in the System Manager
					Options:=, // Not used
					//OUT
					Done=>stAxis.bStopDone,
					Busy=>bStopBusy,
					Active=>bStoping,
					CommandAborted=>bStopCmdAbort,
					Error=>bStopError,
					ErrorID=>udiStopErrorId,
					);

(** HALT **)
	(* mcHalt *)
		mcAxisHalt(
 					//IN
 					Axis:=stAxis.stDriveAx8206.AxisRef,
 					Execute:=stAxis.bHaltExecute,
 					//Deceleration:=, // see the Axis Configuration in the System Manager
 					//Jerk:=, // see the Axis Configuration in the System Manager
 					Options:=, // Not used
 					//OUT
 					Done=>stAxis.bHaltDone,
 					Busy=>bHaltBusy,
 					Active=>bHalting,
 					CommandAborted=>bHaltCmdAbort,
 					Error=>bHaltError,
 					ErrorID=>udiStopErrorId,
					);

(** JOG **)
	(* mcJog *)
		mcAxisJog(
				// IN
				Axis:=stAxis.stDriveAx8206.AxisRef,
				JogForward:=(stAxis.bJogPlus AND stAxis.bJogEnable),
				JogBackwards:=(stAxis.bJogMinus AND stAxis.bJogEnable),
				Mode:=stAxis.eJogMode,
				Position:=stAxis.lrJogPos, // only in Mode INCHING
				Velocity:=stAxis.lrJogVel,
				//Acceleration:=stAxis.rJogAcc, // see the Axis Configuration in the System Manager
				//Deceleration:=stAxis.rJogDec, // see the Axis Configuration in the System Manager
				//Jerk:=rJogJerk, // see the Axis Configuration in the System Manager
				// OUT
				Done=>stAxis.bJogDone,
				Busy=>bJogBusy,
				Active=>bJogging,
				CommandAborted=>bJogCmdAbort,
				Error=>bJogError,
				ErrorID=>udiJogErrorId,
				);

(** AUTO **)
	(* mcMoveAbs *)	
		mcAxisMoveAbs(
					// IN
					Axis:=stAxis.stDriveAx8206.AxisRef,
					Execute:=(stAxis.bAutoCmdAbs AND stAxis.bAutoEnable),
					Position:=stAxis.lrAutoPosAbs,
					Velocity:=stAxis.lrAutoVelAbs,
					//Acceleration:=stAxis.rAutoAccAbs,
					//Deceleration:=stAxis.rAutoDecAbs,
					//Jerk:=stAxis.rAutoJerkAbs,
					//BufferMode:=mcAborting,
					// OUT
					Done=>stAxis.bAutoDone,
					Busy=>bAutoBusy,
					Error=>bAutoError,
					ErrorID=>udiAutoErrorId
					);

(** RESET **)
	IF stAxis.bEventAck AND stAxis.bAlAxisFault THEN
		stAxis.bResetCmd:=TRUE;
	END_IF
	(* mcReset *)
		mcAxisReset(	
					// IN
					Axis:=stAxis.stDriveAx8206.AxisRef,
					Execute:=stAxis.bResetCmd,
					// OUT
					Done=>bResetDone,
					Busy=>bResetBusy,
					Error=>bResetError,
					ErrorID=>udiResetErrorId,
					);
	IF bResetDone OR bResetError THEN
		stAxis.bResetCmd:=FALSE;
	END_IF
	
(** READ BOOL PARAMETER **)	
	mcReadbParameter(
					// IN
					Axis:=stAxis.stDriveAx8206.AxisRef,
					Enable:=stAxis.bReadbEnable,
					ParameterNumber:=stAxis.mcAxisReadParameterb,
					ReadMode:=E_ReadMode.READMODE_CYCLIC,
					// OUT
					Value=>stAxis.bReadbValue,
					Valid=>stAxis.bReadbValid,
					Busy=>bReadbBusy,
					Error=>bReadbError,
					ErrorID=>udiReadbErrorId
					);

(** READ LREAL PARAMETER **)	
	mcReadlrParameter(
					// IN
					Axis:=stAxis.stDriveAx8206.AxisRef,
					Enable:= stAxis.bReadlrEnable,
					ParameterNumber:=stAxis.mcAxisReadParameterlr,
					ReadMode:=E_ReadMode.READMODE_CYCLIC,
					// OUT
					Value=>stAxis.lrReadlrValue,
					Valid=>stAxis.bReadlrValid,
					Busy=>bReadlrBusy,
					Error=>bReadlrError,
					ErrorID=>udiReadlrErrorId
					);

(** WRITE BOOL PARAMETER **)
	mcWritebParameter(
					 // IN
					 Axis:=stAxis.stDriveAx8206.AxisRef,
					 Execute:=stAxis.bWritebExecute,
					 ParameterNumber:=stAxis.mcAxisWriteParameterb,
					 Value:=stAxis.bWritebValue,
					 // OUT
					 Done=>stAxis.bWritebDone,
					 Busy=>stAxis.bWritebBusy,
					 Error=>bWritebError,
					 ErrorID=>udiWritebErrorId
					 );
	
(** WRITE LREAL PARAMETER **)
	mcWritelrParameter(
					 // IN
					 Axis:=stAxis.stDriveAx8206.AxisRef,
					 Execute:=stAxis.bWritelrExecute,
					 ParameterNumber:=stAxis.mcAxisWriteParameterlr,
					 Value:=stAxis.lrWritelrValue,
					 // OUT
					 Done=>stAxis.bWritelrDone,
					 Busy=>stAxis.bWritelrBusy,
					 Error=>bWritelrError,
					 ErrorID=>udiWritelrErrorId
					 );

(** SET POSITION OFFSET (Referencing) **)
	fbSetPositionOffset(
						//IN
						Axis:=stAxis.stDriveAx8206.AxisRef,
						Execute:=stAxis.bSetOffsetExecute,
						Position:=0,
						Relative:=FALSE, // Relative is to add the position at the actual offset (offset=offset+position), but we want to set a new position (offset=position)
						Memory:=E_PositionOffsetMemory.ePositionOffsetMemory_Encoder, // Offset is Set in the Motor Encoder and not in the Drive
						Feedback:=,
						//OUT
						Busy=>bSetPositionOffsetBusy,
						Error=>bSetPositionOffsetError,
						ErrorID=>udiSetPositionOffsetErrorId
						);
 
 (** DELETE POSITION OFFSET (Referencing) **) 
	fbDeletePositionOffset( // = Factory reset of the Axis position 
							//IN
							Axis:=stAxis.stDriveAx8206.AxisRef,
							Execute:=stAxis.bDeleteOffsetExecute,
							Memory:=E_PositionOffsetMemory.ePositionOffsetMemory_Encoder, // Offset is Set in the Motor Encoder and not in the Drive
							Feedback:=,							
							//OUT
							Busy=>bDeletePositionOffsetBusy,
							Error=>bDeletePositionOffsetError,
							ErrorID=>udiDeletePositionOffsetErrorId
							);
 
(** ERROR **)
	bError:=(bPowerError OR bStopError OR bJogError OR bAutoError OR bResetError);
	bErrorParameter:=(bReadlrError OR bReadbError OR bWritelrError OR bWritebError);
	bErrorReferencing:=(bDeletePositionOffsetError OR bSetPositionOffsetError);

END_FUNCTION_BLOCK

// ---- 10_Axes/03_POUs/02_FBs/FB_Handwheel.TcPOU
FUNCTION_BLOCK FB_Handwheel
VAR_INPUT
	(** INT **)
		iHandwheelNumber : INT ; // Number of the handwheel
END_VAR
VAR_OUTPUT
END_VAR
VAR_IN_OUT
	(** ST **)
		stHandwheel : ST_Handwheel ;
END_VAR
VAR
	(** LREAL **)
		lrJogUnitValue : LREAL ; // Unit value for the jog
		lrJogMaxSpeed : LREAL ; // Max Speed for te Jog (in function of the Axis) (mm/s)
		lrJogMaxIncrCycle : LREAL ; // Max Incrément per PLC cycle for Jog
	
	(** DINT **)
		diCounterValueMemory : DINT ; // Memory Value of the Counter
		diDeltaPulses : DINT ; // Delta of the pulses
		diJogMaxPulseCycle : DINT ; // Max Pulse by PLC Cycle
	
	(** FLAG **)
		bChange : BOOL ;
		bJogRequest : BOOL ; // Request for Jog	
		bJogRequestMemory : BOOL ; // Memory Request for Jog	
	
	(** FB **)
		TonPowerON : TON ; // Power timer
		TonPowerOFF : TON ; // Power timer
		TonInactivity : TON ; // Inactivity timer
END_VAR

//-----------------------------------------------------------------------------------------
//
//                  				FB_Handwheel
//
//							Gestion manivelle(s) déportée(s)   			
//-----------------------------------------------------------------------------------------
//
//Auteur: G.GOETZ
//Création: 19.01.2026
//Dernière modification : 19.01.2026 (G.GOETZ)
//       			
//-----------------------------------------------------------------------------------------
//
//     							Liste des modifications  	
//
// 19.01.2026 (G.GOETZ) -> Création		
//-----------------------------------------------------------------------------------------

IF stHandwheel.bPresence AND stHandwheel.bEnable THEN
		
	(** EVENTS **)
	
		
	(** ALARMS **)
		
		
	(** MESSAGES **)
	//Manivelle active
	
	(** SELECTOR **) // GRAY code
		(* Axis X/Y/Z*)
			IF (NOT stHandwheel.bAxisSelectorB0) AND (NOT stHandwheel.bAxisSelectorB1) AND (NOT stHandwheel.bAxisSelectorB2) THEN // 0-0-0
				stHandwheel.eAxisSelect:=ENUM_Axis_Select.X;	
				lrJogMaxSpeed:=GV_Axes.lrJogMaxSpeedAxisX;
			ELSIF stHandwheel.bAxisSelectorB0 AND (NOT stHandwheel.bAxisSelectorB1) AND (NOT stHandwheel.bAxisSelectorB2) THEN // 1-0-0
				stHandwheel.eAxisSelect:=ENUM_Axis_Select.Y;	
				lrJogMaxSpeed:=GV_Axes.lrJogMaxSpeedAxisY;
			ELSIF stHandwheel.bAxisSelectorB0 AND stHandwheel.bAxisSelectorB1 AND (NOT stHandwheel.bAxisSelectorB2) THEN // 1-1-0
				stHandwheel.eAxisSelect:=ENUM_Axis_Select.Z;	
				lrJogMaxSpeed:=GV_Axes.lrJogMaxSpeedAxisZ;
			ELSIF (NOT stHandwheel.bAxisSelectorB0) AND stHandwheel.bAxisSelectorB1 AND (NOT stHandwheel.bAxisSelectorB2) THEN // 0-1-0
				stHandwheel.eAxisSelect:=ENUM_Axis_Select.Arm;	
				lrJogMaxSpeed:=GV_Axes.lrJogMaxSpeedAxisArm;
			ELSE
				stHandwheel.eAxisSelect:=ENUM_Axis_Select.None;
				lrJogMaxSpeed:=0.0;
			END_IF
		(* Incremental x0/x1/x10/x100/x1000*)
			IF (NOT stHandwheel.bIncrSelectorB0) AND (NOT stHandwheel.bIncrSelectorB1) AND (NOT stHandwheel.bIncrSelectorB2) THEN // 0-0-0
				stHandwheel.eIncrSelect:=ENUM_Handwheel_Incr_Select.x0;
				stHandwheel.lrJogVel:=0.0;
				lrJogUnitValue:=0.0;
			ELSIF stHandwheel.bIncrSelectorB0 AND (NOT stHandwheel.bIncrSelectorB1) AND (NOT stHandwheel.bIncrSelectorB2) THEN // 1-0-0
				stHandwheel.eIncrSelect:=ENUM_Handwheel_Incr_Select.x1;
				stHandwheel.lrJogVel:=(lrJogMaxSpeed/1000);
				lrJogUnitValue:=GV_Handwheel.lrUnitIncrx1;
			ELSIF stHandwheel.bIncrSelectorB0 AND stHandwheel.bIncrSelectorB1 AND (NOT stHandwheel.bIncrSelectorB2) THEN // 1-1-0
				stHandwheel.eIncrSelect:=ENUM_Handwheel_Incr_Select.x10;
				stHandwheel.lrJogVel:=(lrJogMaxSpeed/100);
				lrJogUnitValue:=GV_Handwheel.lrUnitIncrx10;
			ELSIF (NOT stHandwheel.bIncrSelectorB0) AND stHandwheel.bIncrSelectorB1 AND (NOT stHandwheel.bIncrSelectorB2) THEN // 0-1-0
				stHandwheel.eIncrSelect:=ENUM_Handwheel_Incr_Select.x100;
				stHandwheel.lrJogVel:=(lrJogMaxSpeed/10);
				lrJogUnitValue:=GV_Handwheel.lrUnitIncrx100;
			ELSIF (NOT stHandwheel.bIncrSelectorB0) AND stHandwheel.bIncrSelectorB1 AND stHandwheel.bIncrSelectorB2 THEN // 0-1-1
				stHandwheel.eIncrSelect:=ENUM_Handwheel_Incr_Select.x1000;
				stHandwheel.lrJogVel:=(lrJogMaxSpeed/1);
				lrJogUnitValue:=GV_Handwheel.lrUnitIncrx1000;
			ELSE
				stHandwheel.eIncrSelect:=ENUM_Handwheel_Incr_Select.Unknow;
				stHandwheel.lrJogVel:=0.0;
				lrJogUnitValue:=0.0;
			END_IF			

	(** POWER **)
		(* Inactivity on the handwheel *)
			IF stHandwheel.bButtonPlus OR stHandwheel.bButtonMinus OR stHandwheel.bButtonFast 
			OR (stHandwheel.eAxisSelect<>stHandwheel.eAxisSelectMemory) OR (stHandwheel.eIncrSelect<>stHandwheel.eIncrSelectMemory)
			OR diDeltaPulses<>0 THEN
				stHandwheel.bActivity:=TRUE;
			ELSE
				stHandwheel.bActivity:=FALSE;
			END_IF
			TonInactivity(IN:=(NOT stHandwheel.bActivity),PT:=GV_Handwheel.tInactivityTime);
		(* ON/OFF *)
			IF (NOT stHandwheel.bButtonPlus) AND (NOT stHandwheel.bButtonMinus) THEN
				bChange:=FALSE;
			END_IF
			TonPowerON(IN:=(stHandwheel.bButtonPlus AND stHandwheel.bButtonMinus AND (NOT stHandwheel.bPower)),PT:=GV_Handwheel.tPowerTime);
			TonPowerOFF(IN:=(stHandwheel.bButtonPlus AND stHandwheel.bButtonMinus AND stHandwheel.bPower),PT:=GV_Handwheel.tPowerTime);
			IF TonPowerON.Q AND (NOT bChange) AND (NOT GV_General.bEmergencyStop) THEN
				stHandwheel.bPower:=TRUE;
				bChange:=TRUE;
			END_IF
			IF (TonPowerOFF.Q AND (NOT bChange))THEN
				stHandwheel.bPower:=FALSE;
				bChange:=TRUE;
			END_IF
			IF TonInactivity.Q OR (NOT GV_General.bSafety) THEN
				stHandwheel.bPower:=FALSE;
			END_IF	
			
	(** CONTER -> PULSE **)
		(* Max Pulse *) 
			diJogMaxPulseCycle:=MAX(1,REAL_TO_DINT(200*MAX(PRG_MAIN.lrLastExecTime_s,0.005))); // 100 pulses/tr -> 2tr/s by the human = 200pulses/s -> Task speed
		(* Ask *)
			IF stHandwheel.bSoftwareGateValid AND stHandwheel.bPower THEN // Counter is allowed
				diDeltaPulses:=(UDINT_TO_DINT(stHandwheel.udiCounterValue)-diCounterValueMemory); // Delta pulses
				diCounterValueMemory:=UDINT_TO_DINT(stHandwheel.udiCounterValue); // Memory
			ELSE
				diDeltaPulses:=0;
				diCounterValueMemory:=UDINT_TO_DINT(stHandwheel.udiCounterValue);
			END_IF
		(* Limit Pulse *)
			IF ABS(diDeltaPulses)>diJogMaxPulseCycle THEN
				diDeltaPulses:=0;
			END_IF	
	
	(** JOG **)
		(* Max Incr *) 
			lrJogMaxIncrCycle:=MIN(lrJogMaxSpeed*PRG_MAIN.lrLastExecTime_s,lrJogUnitValue*DINT_TO_REAL(diJogMaxPulseCycle)); // Max Speed (mm/s) * Task time (s)
		(* Direction *)
			IF diDeltaPulses>0 OR stHandwheel.bButtonPlus AND (NOT stHandwheel.bButtonMinus) THEN
				stHandwheel.eJogDirection:=ENUM_Jog_Direction.Plus;
			ELSIF diDeltaPulses<0 OR (NOT stHandwheel.bButtonPlus) AND stHandwheel.bButtonMinus THEN
				stHandwheel.eJogDirection:=ENUM_Jog_Direction.Minus;
			ELSE
				stHandwheel.eJogDirection:=ENUM_Jog_Direction.None;			
			END_IF
		(* Incremental Request *)
			(*Ask*)
				stHandwheel.lrJogIncrRequest:=0.0;
				IF stHandwheel.bPower AND stHandwheel.eAxisSelect<>ENUM_Axis_Select.None AND stHandwheel.eIncrSelect<>ENUM_Handwheel_Incr_Select.Unknow AND stHandwheel.eJogDirection<>ENUM_Jog_Direction.None THEN
					IF diDeltaPulses<>0 THEN
						stHandwheel.lrJogIncrRequest:=DINT_TO_REAL(diDeltaPulses)*lrJogUnitValue; // +/- X Pulse with the handwheel
						stHandwheel.eJogMode:=ENUM_Jog_Mode.Inching;
					ELSIF stHandwheel.bButtonPlus AND (NOT stHandwheel.bButtonMinus) THEN
						stHandwheel.lrJogIncrRequest:=lrJogUnitValue; // + 1 Pulse with the button
						stHandwheel.eJogMode:=ENUM_Jog_Mode.Inching;
						//stHandwheel.eJogMode:=ENUM_Jog_Mode.Continous;
					ELSIF (NOT stHandwheel.bButtonPlus) AND stHandwheel.bButtonMinus THEN
						stHandwheel.lrJogIncrRequest:=(-lrJogUnitValue); // - 1 Pulse with the button
						stHandwheel.eJogMode:=ENUM_Jog_Mode.Inching;
						//stHandwheel.eJogMode:=ENUM_Jog_Mode.Continous;
					ELSE
						stHandwheel.eJogMode:=ENUM_Jog_Mode.None;
					END_IF		
				ELSE
						stHandwheel.eJogMode:=ENUM_Jog_Mode.None;
				END_IF		
			(*Limit Incr*)
				IF stHandwheel.lrJogIncrRequest>lrJogMaxIncrCycle THEN
					stHandwheel.lrJogIncrRequest:=lrJogMaxIncrCycle;
				END_IF
				IF stHandwheel.lrJogIncrRequest<(-lrJogMaxIncrCycle) THEN
					stHandwheel.lrJogIncrRequest:=(-lrJogMaxIncrCycle);
				END_IF
		(* Request *)
			IF stHandwheel.bPower AND stHandwheel.eAxisSelect<>ENUM_Axis_Select.None AND stHandwheel.eIncrSelect<>ENUM_Handwheel_Incr_Select.Unknow AND stHandwheel.eJogDirection<>ENUM_Jog_Direction.None AND stHandwheel.eJogMode<>ENUM_Jog_Mode.None AND stHandwheel.lrJogIncrRequest<>0 THEN
				bJogRequest:=TRUE;
			ELSE
				bJogRequest:=FALSE;
			END_IF
			(*Rising Edge*)
				stHandwheel.bJogRequestRisingEdge:=(bJogRequest AND (NOT bJogRequestMemory));
				bJogRequestMemory:=bJogRequest;

	(** MEMORY **) // To compare and set the inactivity
		(* Axis Selector *)
			IF stHandwheel.eAxisSelect<>stHandwheel.eAxisSelectMemory THEN
				stHandwheel.eAxisSelectMemory:=stHandwheel.eAxisSelect;
			END_IF
		(* Incremental Selector *)
			IF stHandwheel.eIncrSelect<>stHandwheel.eIncrSelectMemory THEN
				stHandwheel.eIncrSelectMemory:=stHandwheel.eIncrSelect;
			END_IF

ELSE
	(** POWER **)
		(* ON/OFF *)
			stHandwheel.bPower:=FALSE;
END_IF

END_FUNCTION_BLOCK

// ---- 11_CNC/03_POUs/01_PRGs/PRG_CNC.TcPOU
PROGRAM PRG_CNC
VAR
	(** WORD **)
		wSpindleToolLocation : WORD ;	
		wToolToLoadLocation : WORD ;	

	(** BYTE **)
		bSpindleToolLocation1 : BYTE ;	
		bSpindleToolLocation2 : BYTE ;	
		bToolToLoadLocation1 : BYTE ;	
		bToolToLoadLocation2 : BYTE ;
		
	(** FB **)
		fbCncFanuc : FB_CNC_Fanuc ;
		fbCncHeidenhain : FB_CNC_Heidenhain ;
		fbEventGroupAssignement : FB_Event_Group_Number_Assignement ;
END_VAR

//-----------------------------------------------------------------------------------------
//
//                  				PRG_CNC
//
//							Programme partie CNC    			
//-----------------------------------------------------------------------------------------
//
//Auteur: G.GOETZ
//Création: 27.01.2026
//Dernière modification : 27.01.2026 (G.GOETZ)
//       			
//-----------------------------------------------------------------------------------------
//
//     							Liste des modifications  	
//
// 27.01.2026 (G.GOETZ) -> Création	
//-----------------------------------------------------------------------------------------

(** INPUT **)
	(* Byte 0 *)
		GV_CNC.stFanucData.stCncMagazine.biLife:=GV_CNC.stFanucData.stCncMagazine.byi0.0 ; // Life bit -> X0.0
		GV_CNC.stFanucData.stCncMagazine.biToolAnticipation:=GV_CNC.stFanucData.stCncMagazine.byi0.1 ; // Anticipation to prepare the next Tool -> X0.1
		GV_CNC.stFanucData.stCncMagazine.biAllowedOpenIntermediateDoor:=GV_CNC.stFanucData.stCncMagazine.byi0.2 ; // Allowed to open the Intermediate Door 02 -> X0.2
		GV_CNC.stFanucData.stCncMagazine.biLoadUnloadRequest:=GV_CNC.stFanucData.stCncMagazine.byi0.3 ; // Request to Load and Unload a Tool -> X0.3
		GV_CNC.stFanucData.stCncMagazine.biLoadRequest:=GV_CNC.stFanucData.stCncMagazine.byi0.4 ; // Request to only Load a Tool -> X0.4
		GV_CNC.stFanucData.stCncMagazine.biUnloadRequest:=GV_CNC.stFanucData.stCncMagazine.byi0.5 ; // Request to only Unload a Tool -> X0.5
		GV_CNC.stFanucData.stCncMagazine.biLoadUnloadEnd:=GV_CNC.stFanucData.stCncMagazine.byi0.6 ; // End of the Request -> X0.6
		GV_CNC.stFanucData.stCncMagazine.biAllowedCloseIntermediateDoor:=GV_CNC.stFanucData.stCncMagazine.byi0.7 ; // Allowed to close the Intermediate Door 07 -> X0.7
	(* Byte 1 *)
		GV_CNC.stFanucData.stCncMagazine.biInCycle:=GV_CNC.stFanucData.stCncMagazine.byi1.0 ; // CNC in Cycle -> X1.0
		GV_CNC.stFanucData.stCncMagazine.biEvacuateArm:=GV_CNC.stFanucData.stCncMagazine.byi1.1 ; // Request to evacuate the Changing Arm and close the Intermediate Door -> X1.1
		GV_CNC.stFanucData.stCncMagazine.biReserve12:=GV_CNC.stFanucData.stCncMagazine.byi1.2 ; // Reserve 12 -> X1.2
		GV_CNC.stFanucData.stCncMagazine.biReserve13:=GV_CNC.stFanucData.stCncMagazine.byi1.3 ; // Reserve 13 -> X1.3
		GV_CNC.stFanucData.stCncMagazine.biReserve14:=GV_CNC.stFanucData.stCncMagazine.byi1.4 ; // Reserve 14 -> X1.4
		GV_CNC.stFanucData.stCncMagazine.biReserve15:=GV_CNC.stFanucData.stCncMagazine.byi1.5 ; // Reserve 15 -> X1.5
		GV_CNC.stFanucData.stCncMagazine.biReserve16:=GV_CNC.stFanucData.stCncMagazine.byi1.6 ; // Reserve 16 -> X1.6
		GV_CNC.stFanucData.stCncMagazine.biDoorClosed:=GV_CNC.stFanucData.stCncMagazine.byi1.7 ; // CNC Door closed (operator) -> X1.7
	(* Byte 2 *)
		GV_CNC.stFanucData.stCncMagazine.biEmergencyStop:=(NOT GV_CNC.stFanucData.stCncMagazine.byi2.0) ; // Emergency Stop -> X2.0
		GV_CNC.stFanucData.stCncMagazine.biPower:=GV_CNC.stFanucData.stCncMagazine.byi2.1 ; // Power -> X2.1
		GV_CNC.stFanucData.stCncMagazine.biAir:=GV_CNC.stFanucData.stCncMagazine.byi2.2 ; // Air -> X2.2
		GV_CNC.stFanucData.stCncMagazine.biShutdown:=GV_CNC.stFanucData.stCncMagazine.byi2.3 ; // Shutdown -> X2.3
		GV_CNC.stFanucData.stCncMagazine.biReserve24:=GV_CNC.stFanucData.stCncMagazine.byi2.4 ; // Reserve 24 -> X2.4
		GV_CNC.stFanucData.stCncMagazine.biReserve25:=GV_CNC.stFanucData.stCncMagazine.byi2.5 ; // Reserve 25 -> X2.5
		GV_CNC.stFanucData.stCncMagazine.biReserve26:=GV_CNC.stFanucData.stCncMagazine.byi2.6 ; // Reserve 26 -> X2.6
		GV_CNC.stFanucData.stCncMagazine.biReserve27:=GV_CNC.stFanucData.stCncMagazine.byi2.7 ; // Reserve 27 -> X2.7
	(* Byte 3 *)
		GV_CNC.stFanucData.stCncMagazine.biReserve30:=GV_CNC.stFanucData.stCncMagazine.byi3.0 ; // Reserve 30 -> X3.0
		GV_CNC.stFanucData.stCncMagazine.biReserve31:=GV_CNC.stFanucData.stCncMagazine.byi3.1 ; // Reserve 31 -> X3.1
		GV_CNC.stFanucData.stCncMagazine.biReserve32:=GV_CNC.stFanucData.stCncMagazine.byi3.2 ; // Reserve 32 -> X3.2
		GV_CNC.stFanucData.stCncMagazine.biReserve33:=GV_CNC.stFanucData.stCncMagazine.byi3.3 ; // Reserve 33 -> X3.3
		GV_CNC.stFanucData.stCncMagazine.biReserve34:=GV_CNC.stFanucData.stCncMagazine.byi3.4 ; // Reserve 34 -> X3.4
		GV_CNC.stFanucData.stCncMagazine.biReserve35:=GV_CNC.stFanucData.stCncMagazine.byi3.5 ; // Reserve 35 -> X3.5
		GV_CNC.stFanucData.stCncMagazine.biReserve36:=GV_CNC.stFanucData.stCncMagazine.byi3.6 ; // Reserve 36 -> X3.6
		GV_CNC.stFanucData.stCncMagazine.biReserve37:=GV_CNC.stFanucData.stCncMagazine.byi3.7 ; // Reserve 37 -> X3.7
	(* Byte 4 *)
		GV_CNC.stFanucData.stCncMagazine.biReserve40:=GV_CNC.stFanucData.stCncMagazine.byi4.0 ; // Reserve 40 -> X4.0
		GV_CNC.stFanucData.stCncMagazine.biReserve41:=GV_CNC.stFanucData.stCncMagazine.byi4.1 ; // Reserve 41 -> X4.1
		GV_CNC.stFanucData.stCncMagazine.biReserve42:=GV_CNC.stFanucData.stCncMagazine.byi4.2 ; // Reserve 42 -> X4.2
		GV_CNC.stFanucData.stCncMagazine.biReserve43:=GV_CNC.stFanucData.stCncMagazine.byi4.3 ; // Reserve 43 -> X3.3
		GV_CNC.stFanucData.stCncMagazine.biReserve44:=GV_CNC.stFanucData.stCncMagazine.byi4.4 ; // Reserve 44 -> X4.4
		GV_CNC.stFanucData.stCncMagazine.biReserve45:=GV_CNC.stFanucData.stCncMagazine.byi4.5 ; // Reserve 45 -> X4.5
		GV_CNC.stFanucData.stCncMagazine.biReserve46:=GV_CNC.stFanucData.stCncMagazine.byi4.6 ; // Reserve 46 -> X4.6
		GV_CNC.stFanucData.stCncMagazine.biReserve47:=GV_CNC.stFanucData.stCncMagazine.byi4.7 ; // Reserve 47 -> X4.7
	(* Byte 5 *)
		GV_CNC.stFanucData.stCncMagazine.biReserve50:=GV_CNC.stFanucData.stCncMagazine.byi5.0 ; // Reserve 50 -> X5.0
		GV_CNC.stFanucData.stCncMagazine.biReserve51:=GV_CNC.stFanucData.stCncMagazine.byi5.1 ; // Reserve 51 -> X5.1
		GV_CNC.stFanucData.stCncMagazine.biReserve52:=GV_CNC.stFanucData.stCncMagazine.byi5.2 ; // Reserve 52 -> X5.2
		GV_CNC.stFanucData.stCncMagazine.biReserve53:=GV_CNC.stFanucData.stCncMagazine.byi5.3 ; // Reserve 53 -> X5.3
		GV_CNC.stFanucData.stCncMagazine.biReserve54:=GV_CNC.stFanucData.stCncMagazine.byi5.4 ; // Reserve 54 -> X5.4
		GV_CNC.stFanucData.stCncMagazine.biReserve55:=GV_CNC.stFanucData.stCncMagazine.byi5.5 ; // Reserve 55 -> X5.5
		GV_CNC.stFanucData.stCncMagazine.biReserve56:=GV_CNC.stFanucData.stCncMagazine.byi5.6 ; // Reserve 56 -> X5.6
		GV_CNC.stFanucData.stCncMagazine.biReserve57:=GV_CNC.stFanucData.stCncMagazine.byi5.7 ; // Reserve 57 -> X5.7
	(* Byte 6 *)
		GV_CNC.stFanucData.iSpindleToolType:=BYTE_TO_INT(GV_CNC.stFanucData.stCncMagazine.byiSpindleToolType) ;
	(* Byte 7 *)
		GV_CNC.stFanucData.iToolToLoadType:=BYTE_TO_INT(GV_CNC.stFanucData.stCncMagazine.byiToolToLoadType) ;
	(* Byte 8-9 *)
		wSpindleToolLocation:=GV_CNC.stFanucData.stCncMagazine.wiSpindleToolLocation;
		//MSB  
		bSpindleToolLocation1:=WORD_TO_BYTE(SHR(wSpindleToolLocation,8));
		//LSB
		bSpindleToolLocation2:=WORD_TO_BYTE(wSpindleToolLocation AND 16#FF);
		wSpindleToolLocation:=(SHL(BYTE_TO_WORD(bSpindleToolLocation2),8) OR BYTE_TO_WORD(bSpindleToolLocation1));

		GV_CNC.stFanucData.iSpindleToolLocation:=WORD_TO_INT(wSpindleToolLocation) ;
	(* Byte 10-11 *)
		wToolToLoadLocation:=GV_CNC.stFanucData.stCncMagazine.wiToolToLoadLocation;
		//MSB  
		bToolToLoadLocation1:=WORD_TO_BYTE(SHR(wToolToLoadLocation,8));
		//LSB
		bToolToLoadLocation2:=WORD_TO_BYTE(wToolToLoadLocation AND 16#FF);
		wToolToLoadLocation:=(SHL(BYTE_TO_WORD(bToolToLoadLocation2),8) OR BYTE_TO_WORD(bToolToLoadLocation1));
	
		GV_CNC.stFanucData.iToolToLoadLocation:=WORD_TO_INT(wToolToLoadLocation) ;

(** SETUP **)
	GV_CNC.bPresence:=TRUE; // CNC prensence or not
	(* Enable *)
		IF GV_HMI.rtCNCEnable.Q THEN
			IF (NOT GV_CNC.bEnable) THEN
				GV_CNC.bEnable:=TRUE;
			ELSE
				GV_CNC.bEnable:=FALSE;
			END_IF
		END_IF
		//GV_CNC.bEnable:=TRUE;
	GV_CNC.bFocas:=TRUE; // With Focas or not
	fbEventGroupAssignement(iEventGroup:=GV_CNC.iEventGroup);
	GV_CNC.bEventAck:=GV_HMI.bEventAck; // Events Acknowledgement
	GV_CNC.eType:=ENUM_CNC_type.Fanuc; // CNC type
	// ...

(** PROCESS **)
	(* Air blow *)
	IF (NOT GV_General.bSafety) OR (NOT GV_General.bAir) OR ((GV_OpMode.eOpMode=ENUM_OpMode.AUTO AND (NOT GV_Cycle.bStartStop)) OR GV_OpMode.eOpMode<>ENUM_OpMode.AUTO) THEN
		GV_CNC.stFanucData.stMagazineCNC.boAirBlowIntermediateDoor:=FALSE;
	END_IF

(** SPINDLE **)
	(*Memory*)
		IF (GV_CNC.stSpindle.iAbsLocationNumberMemory>0 AND GV_CNC.stSpindle.iRelLocationNumberMemory>0) THEN
			GV_CNC.stSpindle.bToolPresenceMemory:=TRUE;
		ELSE
			GV_CNC.stSpindle.bToolPresenceMemory:=FALSE;
		END_IF
		
(** FB_CNC_xxx **)
	CASE GV_CNC.eType OF
		ENUM_CNC_Type.Fanuc:
			fbCncFanuc(StCncData:=GV_CNC.stFanucData);
		ENUM_CNC_Type.Heidenhain:
			fbCncHeidenhain(StCncData:=GV_CNC.stHeidenhainData);
	END_CASE

(** OUTPUT **)
	(* Byte 0 *)
		GV_CNC.stFanucData.stMagazineCNC.byo0.0:=GV_CNC.stFanucData.stMagazineCNC.boLife; // Magazine Life bit -> X0.0
		GV_CNC.stFanucData.stMagazineCNC.byo0.1:=GV_CNC.stFanucData.stMagazineCNC.boToolAnticipated; // Next tool is prepared/anticipated -> X0.1
		GV_CNC.stFanucData.stMagazineCNC.byo0.2:=GV_CNC.stFanucData.stMagazineCNC.boReserve02; // Reserve 02 -> X0.2
		GV_CNC.stFanucData.stMagazineCNC.byo0.3:=GV_CNC.stFanucData.stMagazineCNC.boReserve03; // Reserve 03 -> X0.3
		GV_CNC.stFanucData.stMagazineCNC.byo0.4:=GV_CNC.stFanucData.stMagazineCNC.boReserve04; // Reserve 04 -> X0.4
		GV_CNC.stFanucData.stMagazineCNC.byo0.5:=GV_CNC.stFanucData.stMagazineCNC.boReserve05; // Reserve 05 -> X0.5
		GV_CNC.stFanucData.stMagazineCNC.byo0.6:=GV_CNC.stFanucData.stMagazineCNC.boArmInCncPosition; // Loading Arm in position in the CNC -> X0.6
		GV_CNC.stFanucData.stMagazineCNC.byo0.7:=GV_CNC.stFanucData.stMagazineCNC.boNoFault; // No Fault on the Magazine -> X0.7
	(* Byte 1 *)
		GV_CNC.stFanucData.stMagazineCNC.byo1.0:=GV_CNC.stFanucData.stMagazineCNC.boArmOutOfCncArea; // Changing Arm out of Cnc area -> X1.0
		GV_CNC.stFanucData.stMagazineCNC.byo1.1:=GV_CNC.stFanucData.stMagazineCNC.boOpenManipulatorGripper; // Open the manipulator gripper -> X1.1
		GV_CNC.stFanucData.stMagazineCNC.byo1.2:=GV_CNC.stFanucData.stMagazineCNC.boAirBlowIntermediateDoor; // Air blow of the Intermediate Door -> X1.2
		GV_CNC.stFanucData.stMagazineCNC.byo1.3:=GV_CNC.stFanucData.stMagazineCNC.boIntermediateDoorOpen; // Intermediate Door is open -> X1.3
		GV_CNC.stFanucData.stMagazineCNC.byo1.4:=GV_CNC.stFanucData.stMagazineCNC.boIntermediateDoorClose; // Intermediate Door is close -> X1.4
		GV_CNC.stFanucData.stMagazineCNC.byo1.5:=GV_CNC.stFanucData.stMagazineCNC.boReserve15; // Reserve 15 -> X1.5
		GV_CNC.stFanucData.stMagazineCNC.byo1.6:=GV_CNC.stFanucData.stMagazineCNC.boReserve16; // Reserve 16 -> X1.6
		GV_CNC.stFanucData.stMagazineCNC.byo1.7:=GV_CNC.stFanucData.stMagazineCNC.boReserve17; // Reserve 17 -> X1.7
	(* Byte 2 *)
		GV_CNC.stFanucData.stMagazineCNC.byo2.0:=GV_CNC.stFanucData.stMagazineCNC.boReserve20; // Reserve 20 -> X2.0
		GV_CNC.stFanucData.stMagazineCNC.byo2.1:=GV_CNC.stFanucData.stMagazineCNC.boReserve21; // Reserve 21 -> X2.1
		GV_CNC.stFanucData.stMagazineCNC.byo2.2:=GV_CNC.stFanucData.stMagazineCNC.boReserve22; // Reserve 22 -> X2.2
		GV_CNC.stFanucData.stMagazineCNC.byo2.3:=GV_CNC.stFanucData.stMagazineCNC.boReserve23; // Reserve 23 -> X2.3
		GV_CNC.stFanucData.stMagazineCNC.byo2.4:=GV_CNC.stFanucData.stMagazineCNC.boReserve24; // Reserve 24 -> X2.4
		GV_CNC.stFanucData.stMagazineCNC.byo2.5:=GV_CNC.stFanucData.stMagazineCNC.boReserve25; // Reserve 25 -> X2.5
		GV_CNC.stFanucData.stMagazineCNC.byo2.6:=GV_CNC.stFanucData.stMagazineCNC.boReserve26; // Reserve 26 -> X2.6
		GV_CNC.stFanucData.stMagazineCNC.byo2.7:=GV_CNC.stFanucData.stMagazineCNC.boReserve27; // Reserve 27 -> X2.7
	(* Byte 3 *)
		GV_CNC.stFanucData.stMagazineCNC.byo3.0:=GV_CNC.stFanucData.stMagazineCNC.boReserve30; // Reserve 30 -> X3.0
		GV_CNC.stFanucData.stMagazineCNC.byo3.1:=GV_CNC.stFanucData.stMagazineCNC.boReserve31; // Reserve 31 -> X3.1
		GV_CNC.stFanucData.stMagazineCNC.byo3.2:=GV_CNC.stFanucData.stMagazineCNC.boReserve32; // Reserve 32 -> X3.2
		GV_CNC.stFanucData.stMagazineCNC.byo3.3:=GV_CNC.stFanucData.stMagazineCNC.boReserve33; // Reserve 33 -> X3.3
		GV_CNC.stFanucData.stMagazineCNC.byo3.4:=GV_CNC.stFanucData.stMagazineCNC.boReserve34; // Reserve 34 -> X3.4
		GV_CNC.stFanucData.stMagazineCNC.byo3.5:=GV_CNC.stFanucData.stMagazineCNC.boReserve35; // Reserve 35 -> X3.5
		GV_CNC.stFanucData.stMagazineCNC.byo3.6:=GV_CNC.stFanucData.stMagazineCNC.boReserve36; // Reserve 36 -> X3.6
		GV_CNC.stFanucData.stMagazineCNC.byo3.7:=GV_CNC.stFanucData.stMagazineCNC.boReserve37; // Reserve 37 -> X3.7
	(* Byte 4 *)
		GV_CNC.stFanucData.stMagazineCNC.byo4.0:=GV_CNC.stFanucData.stMagazineCNC.boReserve40; // Reserve 40 -> X4.0
		GV_CNC.stFanucData.stMagazineCNC.byo4.1:=GV_CNC.stFanucData.stMagazineCNC.boReserve41; // Reserve 41 -> X4.1
		GV_CNC.stFanucData.stMagazineCNC.byo4.2:=GV_CNC.stFanucData.stMagazineCNC.boReserve42; // Reserve 42 -> X4.2
		GV_CNC.stFanucData.stMagazineCNC.byo4.3:=GV_CNC.stFanucData.stMagazineCNC.boReserve43; // Reserve 43 -> X4.3
		GV_CNC.stFanucData.stMagazineCNC.byo4.4:=GV_CNC.stFanucData.stMagazineCNC.boReserve44; // Reserve 44 -> X4.4
		GV_CNC.stFanucData.stMagazineCNC.byo4.5:=GV_CNC.stFanucData.stMagazineCNC.boReserve45; // Reserve 45 -> X4.5
		GV_CNC.stFanucData.stMagazineCNC.byo4.6:=GV_CNC.stFanucData.stMagazineCNC.boReserve46; // Reserve 46 -> X4.6
		GV_CNC.stFanucData.stMagazineCNC.byo4.7:=GV_CNC.stFanucData.stMagazineCNC.boReserve47; // Reserve 47 -> X4.7
	(* Byte 5 *)
		GV_CNC.stFanucData.stMagazineCNC.byo5.0:=GV_CNC.stFanucData.stMagazineCNC.boReserve50; // Reserve 50 -> X5.0
		GV_CNC.stFanucData.stMagazineCNC.byo5.1:=GV_CNC.stFanucData.stMagazineCNC.boReserve51; // Reserve 51 -> X5.1
		GV_CNC.stFanucData.stMagazineCNC.byo5.2:=GV_CNC.stFanucData.stMagazineCNC.boReserve52; // Reserve 52 -> X5.2
		GV_CNC.stFanucData.stMagazineCNC.byo5.3:=GV_CNC.stFanucData.stMagazineCNC.boReserve53; // Reserve 53 -> X5.3
		GV_CNC.stFanucData.stMagazineCNC.byo5.4:=GV_CNC.stFanucData.stMagazineCNC.boReserve54; // Reserve 54 -> X5.4
		GV_CNC.stFanucData.stMagazineCNC.byo5.5:=GV_CNC.stFanucData.stMagazineCNC.boReserve55; // Reserve 55 -> X5.5
		GV_CNC.stFanucData.stMagazineCNC.byo5.6:=GV_CNC.stFanucData.stMagazineCNC.boReserve56; // Reserve 56 -> X5.6
		GV_CNC.stFanucData.stMagazineCNC.byo5.7:=GV_CNC.stFanucData.stMagazineCNC.boReserve57; // Reserve 57 -> X5.7

END_PROGRAM

// ---- 11_CNC/03_POUs/02_FBs/FB_CNC_Fanuc.TcPOU
FUNCTION_BLOCK FB_CNC_Fanuc
VAR_INPUT
	(** INT **)
END_VAR
VAR_OUTPUT
END_VAR
VAR_IN_OUT
	(** ST **)
	stCncData : ST_CNC_Fanuc_Data ;
END_VAR
VAR
	(** FB **)
	fbInitEvents : FB_Init_Events ;
	fbEventHMI : FB_Event_HMI ;
	fbLifeBlink : FB_Blink ;
		tonLifeON : TON ;
		tonLifeOFF : TON ;
	tonCommunicationFault : TON ;
END_VAR

//-----------------------------------------------------------------------------------------
//
//                  				FB_CNC_Fanuc
//
//								Gestion CNC Fanuc    			
//-----------------------------------------------------------------------------------------
//
//Auteur: G.GOETZ
//Création: 27.01.2026
//Dernière modification : 27.01.2026 (G.GOETZ)
//       			
//-----------------------------------------------------------------------------------------
//
//     							Liste des modifications  	
//
// 27.01.2026 (G.GOETZ) -> Création	
//-----------------------------------------------------------------------------------------

IF GV_CNC.bPresence THEN
		
	(** EVENTS **)
		IF GV_General.bFirstCycleTask OR GV_General.bFirstCycleSimu THEN
			(*Call first Event because we need to call one Event in the GUID to have it into .xml file*)
			GV_Events.aEventGroup[GV_CNC.iEventGroup].aAlarm[1].fbAlarm.CreateEx(TC_Events.CncFanucAlarms.Alarm1,TRUE,0);
			GV_Events.aEventGroup[GV_CNC.iEventGroup].aOpMessage[1].fbAlarm.CreateEx(TC_Events.CncFanucOpMessages.Message1,TRUE,0);	
			fbInitEvents(iEventGroup:=GV_CNC.iEventGroup,strEventType:='ALARM',strEventGuid:='74BEA104-88D1-4E3B-ADCF-A7B9330EA49F',tcEventSeverity:=2);
			fbInitEvents(iEventGroup:=GV_CNC.iEventGroup,strEventType:='OpMESSAGE',strEventGuid:='30ABA539-286A-4F70-B3DD-90F6994B0D83',tcEventSeverity:=1);
		END_IF
	
	(** ALARMS **)
		(* Life bit *)
				fbLifeBlink(tTimerValue:=T#500MS,bOut=>GV_CNC.stFanucData.stMagazineCNC.boLife); // Life bit Magazine->CNC
			(*Fault*)
				tonLifeON(IN:=GV_CNC.stFanucData.stCncMagazine.biLife,PT:=T#1000MS); // Life bit fault CNC->Magazine
				tonLifeOFF(IN:=(NOT GV_CNC.stFanucData.stCncMagazine.biLife),PT:=T#1000MS); // Life bit fault CNC->Magazine
			(*Reset Fault = Ack*)
				IF GV_CNC.bEventAck THEN
					GV_CNC.bAlLife:=FALSE;
				END_IF
			(*Set Fault*)
				IF (tonLifeON.Q OR tonLifeOFF.Q) AND GV_CNC.bEnable=TRUE THEN
					GV_CNC.bAlLife:=TRUE;
				END_IF
			(*Alarm 1 = Life bit fault*)	
				IF GV_CNC.bAlLife THEN
					GV_Events.aEventGroup[GV_CNC.iEventGroup].aAlarm[1].fbAlarm.ipArguments.Clear();
					fbEventHMI(iEventGroup:=GV_CNC.iEventGroup,iIdEvent:=1,strEventType:='ALARM',bEventSet:=TRUE);
				ELSE
					fbEventHMI(iEventGroup:=GV_CNC.iEventGroup,iIdEvent:=1,strEventType:='ALARM',bEventSet:=FALSE);
				END_IF

		(* Communication *)
			(*Fault*)
				GV_CNC.iCommunicationStatus:=BOOL_TO_INT(GV_CNC.bAlLife); // Life bit fault = Communication fault
				tonCommunicationFault(IN:=GV_CNC.iCommunicationStatus<>0,PT:=T#2000MS); // Communication fault CNC<->Magazine
			(*Reset Fault = Ack*)
				IF GV_CNC.bEventAck THEN
					GV_CNC.bAlCommunication:=FALSE;
				END_IF
			(*Set Fault*)
				IF tonCommunicationFault.Q AND GV_CNC.bEnable=TRUE THEN
					GV_CNC.bAlCommunication:=TRUE;
				END_IF
			(*Alarm 2 = Communication fault*)	
				IF GV_CNC.bAlCommunication THEN
					GV_Events.aEventGroup[GV_CNC.iEventGroup].aAlarm[2].fbAlarm.ipArguments.Clear();
					fbEventHMI(iEventGroup:=GV_CNC.iEventGroup,iIdEvent:=2,strEventType:='ALARM',bEventSet:=TRUE);
				ELSE
					fbEventHMI(iEventGroup:=GV_CNC.iEventGroup,iIdEvent:=2,strEventType:='ALARM',bEventSet:=FALSE);
				END_IF

		(* Emergency Stop *)
			(*Reset Fault = Ack*)
				IF GV_CNC.bEventAck THEN
					GV_CNC.bAlEmergencyStop:=FALSE;
				END_IF
			(*Set Fault*)
				IF GV_CNC.stFanucData.stCncMagazine.biEmergencyStop AND GV_CNC.bEnable=TRUE THEN
					GV_CNC.bAlEmergencyStop:=TRUE;
				END_IF
			(*Alarm 3 = External emergency stop fault*)	
				IF GV_CNC.bAlEmergencyStop THEN
					GV_Events.aEventGroup[GV_CNC.iEventGroup].aAlarm[3].fbAlarm.ipArguments.Clear();
					fbEventHMI(iEventGroup:=GV_CNC.iEventGroup,iIdEvent:=3,strEventType:='ALARM',bEventSet:=TRUE);
				ELSE
					fbEventHMI(iEventGroup:=GV_CNC.iEventGroup,iIdEvent:=3,strEventType:='ALARM',bEventSet:=FALSE);
				END_IF

		(* In Fault *)
			(*Reset Fault = Ack*)
				IF GV_CNC.bEventAck THEN
					GV_CNC.bAlCncFault:=FALSE;
				END_IF
			(*Set Fault*)
				IF GV_Events.aEventGroup[GV_CNC.iEventGroup].bAlarmPresence AND GV_CNC.bEnable=TRUE THEN
					GV_CNC.bAlCncFault:=TRUE;
				END_IF
			(*Alarm 4 = CNC in fault*)	
				IF GV_CNC.bAlCncFault THEN
					GV_Events.aEventGroup[GV_CNC.iEventGroup].aAlarm[4].fbAlarm.ipArguments.Clear();
					fbEventHMI(iEventGroup:=GV_CNC.iEventGroup,iIdEvent:=4,strEventType:='ALARM',bEventSet:=TRUE);
				ELSE
					fbEventHMI(iEventGroup:=GV_CNC.iEventGroup,iIdEvent:=4,strEventType:='ALARM',bEventSet:=FALSE);
				END_IF
			
		(* No Air *)
			(*Reset Fault = Ack*)
				IF GV_CNC.bEventAck THEN
					GV_CNC.bAlNoAir:=FALSE;
				END_IF
			(*Set Fault*)
				IF (NOT GV_CNC.stFanucData.stCncMagazine.biAir) AND GV_CNC.bEnable=TRUE THEN
					GV_CNC.bAlNoAir:=TRUE;
				END_IF
			(*Alarm 5 = No air fault*)	
				IF GV_CNC.bAlNoAir THEN
					GV_Events.aEventGroup[GV_CNC.iEventGroup].aAlarm[5].fbAlarm.ipArguments.Clear();
					fbEventHMI(iEventGroup:=GV_CNC.iEventGroup,iIdEvent:=5,strEventType:='ALARM',bEventSet:=TRUE);
				ELSE
					fbEventHMI(iEventGroup:=GV_CNC.iEventGroup,iIdEvent:=5,strEventType:='ALARM',bEventSet:=FALSE);
				END_IF

		(* No Power *)
			(*Reset Fault = Ack*)
				IF GV_CNC.bEventAck THEN
					GV_CNC.bAlNoPower:=FALSE;
				END_IF
			(*Set Fault*)
				IF (NOT GV_CNC.stFanucData.stCncMagazine.biPower) AND GV_CNC.bEnable=TRUE THEN
					GV_CNC.bAlNoPower:=TRUE;
				END_IF
			(*Alarm 6 = No power fault*)	
				IF GV_CNC.bAlNoPower THEN
					GV_Events.aEventGroup[GV_CNC.iEventGroup].aAlarm[6].fbAlarm.ipArguments.Clear();
					fbEventHMI(iEventGroup:=GV_CNC.iEventGroup,iIdEvent:=6,strEventType:='ALARM',bEventSet:=TRUE);
				ELSE
					fbEventHMI(iEventGroup:=GV_CNC.iEventGroup,iIdEvent:=6,strEventType:='ALARM',bEventSet:=FALSE);
				END_IF
			
		(* Focas Fault *)
			(*Reset Fault = Ack*)
				IF GV_CNC.bEventAck THEN
					GV_CNC.bAlFocas:=FALSE;
				END_IF
			(*Set Fault*)//-> Set in Focas
				//IF FALSE AND GV_CNC.bEnable=TRUE THEN
				//	GV_CNC.bAlFocas:=TRUE;
				//END_IF
			(*Alarm 7 = Focas fault*)	
				IF GV_CNC.bAlFocas THEN
					GV_Events.aEventGroup[GV_CNC.iEventGroup].aAlarm[7].fbAlarm.ipArguments.Clear();
					fbEventHMI(iEventGroup:=GV_CNC.iEventGroup,iIdEvent:=7,strEventType:='ALARM',bEventSet:=TRUE);
				ELSE
					fbEventHMI(iEventGroup:=GV_CNC.iEventGroup,iIdEvent:=7,strEventType:='ALARM',bEventSet:=FALSE);
				END_IF
	
	(** OpMESSAGES **)
		(* CNC Not Ready *)
			(*Set/Reset*)
				IF (NOT GV_Events.aEventGroup[GV_CNC.iEventGroup].bAlarmPresence) THEN
					GV_CNC.bReady:=TRUE;
				END_IF
			(*Message 1 = Not ready*)
				IF (NOT GV_CNC.bReady) AND GV_CNC.bEnable=TRUE THEN
					GV_Events.aEventGroup[GV_CNC.iEventGroup].aOpMessage[1].fbAlarm.ipArguments.Clear();
					fbEventHMI(iEventGroup:=GV_CNC.iEventGroup,iIdEvent:=1,strEventType:='OpMESSAGE',bEventSet:=TRUE);
				ELSE
					fbEventHMI(iEventGroup:=GV_CNC.iEventGroup,iIdEvent:=1,strEventType:='OpMESSAGE',bEventSet:=FALSE);
				END_IF
			
		(* CNC Not In Cycle *)
			(*Message 2 = Not in cycle*)
				IF (NOT GV_CNC.stFanucData.stCncMagazine.biInCycle) AND GV_CNC.bEnable=TRUE THEN
					GV_Events.aEventGroup[GV_CNC.iEventGroup].aOpMessage[2].fbAlarm.ipArguments.Clear();
					//fbEventHMI(iEventGroup:=GV_CNC.iEventGroup,iIdEvent:=2,strEventType:='OpMESSAGE',bEventSet:=TRUE);
				ELSE
					fbEventHMI(iEventGroup:=GV_CNC.iEventGroup,iIdEvent:=2,strEventType:='OpMESSAGE',bEventSet:=FALSE);
				END_IF
				
		(* CNC en cycle *)
			(*Message 3 = In cycle*)
				IF GV_CNC.stFanucData.stCncMagazine.biInCycle AND GV_CNC.bEnable=TRUE THEN
					GV_Events.aEventGroup[GV_CNC.iEventGroup].aOpMessage[3].fbAlarm.ipArguments.Clear();
					//fbEventHMI(iEventGroup:=GV_CNC.iEventGroup,iIdEvent:=3,strEventType:='OpMESSAGE',bEventSet:=TRUE);
				ELSE
					fbEventHMI(iEventGroup:=GV_CNC.iEventGroup,iIdEvent:=3,strEventType:='OpMESSAGE',bEventSet:=FALSE);
				END_IF
			
		(* Alarm present *)
			//fbEventHMI.M_Event_Group_State(iEventGroup:=GV_CNC.iEventGroup,bEventPresence=>GV_Events.aEventGroup[GV_CNC.iEventGroup].bAlarmPresence);
			
	(** CNC MANAGEMENT **)
	
		(* Output *)
			GV_CNC.stFanucData.stMagazineCNC.boToolAnticipated:=(GV_CNC.stFanucData.stCncMagazine.biToolAnticipation AND GV_Cycle.bAnticipateLoadDone); // Next tool is prepared/anticipated -> X0.1
			GV_CNC.stFanucData.stMagazineCNC.boArmInCncPosition:=GV_Tool_Magazine.stArm.ePositionAxis=ENUM_Position_Axis.CNC; // Loading Arm in position in the CNC -> X0.6
			GV_CNC.stFanucData.stMagazineCNC.boNoFault:=(NOT GV_HMI.bAlarm); // No Fault on the Magazine -> X0.7
			
// 			IF GV_Tool_Magazine.stArm.lrArmPosition<=(GV_Tool_Magazine.stArm.lrArmManipulator+GV_Tool_Magazine.stArm.lrArmPositionTol) THEN  //(GV_Tool_Magazine.stArm.ePositionAxis=ENUM_Position_Axis.Home OR GV_Tool_Magazine.stArm.ePositionAxis=ENUM_Position_Axis.Work1);
// 				GV_CNC.stFanucData.stMagazineCNC.boArmOutOfCncArea:=TRUE;// Changing Arm out of Cnc area -> X1.0
// 			ELSE
// 				GV_CNC.stFanucData.stMagazineCNC.boArmOutOfCncArea:=FALSE;// Changing Arm out of Cnc area -> X1.0
// 			END_IF
			GV_CNC.stFanucData.stMagazineCNC.boArmOutOfCncArea:=GV_Tool_Magazine.stArm.lrArmPosition<=(GV_Tool_Magazine.stArm.lrArmManipulator+GV_Tool_Magazine.stArm.lrArmPositionTol);
			GV_CNC.stFanucData.stMagazineCNC.boIntermediateDoorOpen:=GV_Cyltronic.aId[1].bWorkPositionDone AND GV_IO.diIntermediateDoorNotClosed; // Intermediate Door is open -> X1.3
			GV_CNC.stFanucData.stMagazineCNC.boIntermediateDoorClose:=(NOT GV_IO.diIntermediateDoorNotClosed); // Intermediate Door is close -> X1.4
			
END_IF

END_FUNCTION_BLOCK

// ---- 11_CNC/03_POUs/02_FBs/FB_CNC_Heidenhain.TcPOU
FUNCTION_BLOCK FB_CNC_Heidenhain
VAR_INPUT
	(** INT **)
END_VAR
VAR_OUTPUT
END_VAR
VAR_IN_OUT
	(** ST **)
	stCncData : ST_CNC_Heidenhain_Data ;
END_VAR
VAR
	(** FB **)
	fbInitEvents : FB_Init_Events ;
	fbEventHMI : FB_Event_HMI ;
	fbLifeBlink : FB_Blink ;
		tonLifeON : TON ;
		tonLifeOFF : TON ;
END_VAR

//-----------------------------------------------------------------------------------------
//
//                  				FB_CNC_Heidenhain
//
//								Gestion CNC Heidenhain    			
//-----------------------------------------------------------------------------------------
//
//Auteur: G.GOETZ
//Création: 27.01.2026
//Dernière modification : 27.01.2026 (G.GOETZ)
//       			
//-----------------------------------------------------------------------------------------
//
//     							Liste des modifications  	
//
// 27.01.2026 (G.GOETZ) -> Création	
//-----------------------------------------------------------------------------------------

IF GV_CNC.bPresence THEN
		
//	(** EVENTS **)
//		(* Init on FirstCycle *)
//			IF GV_General.bFirstCycleTask OR GV_General.bFirstCycleSimu THEN
//				(*Call first Event because we need to call one Event in the GUID to have it into .xml file*)
//				GV_Events.aEventGroup[GV_CNC.iEventGroup].aAlarm[1].fbAlarm.CreateEx(TC_Events.CncFanucAlarms.Alarm1,TRUE,0);
//				GV_Events.aEventGroup[GV_CNC.iEventGroup].aOpMessage[1].fbAlarm.CreateEx(TC_Events.CncFanucOpMessages.Message1,TRUE,0);	
//				fbInitEvents(iEventGroup:=GV_Events.iEventGroupGeneralEvent, strEventType:='ALARM', strEventGuid:='8530B2D2-E45D-443A-863F-6CD9B6401CBE', tcEventSeverity:=2);
//				fbInitEvents(iEventGroup:=GV_Events.iEventGroupGeneralEvent, strEventType:='OpMESSAGE', strEventGuid:='203DF915-0E17-41A7-9E70-D7D6B508BD1C', tcEventSeverity:=1);
//			END_IF
	
//	(** ALARMS **)
//		(* Acknowledgement *)
//		GV_CNC.bEventAck:=GV_HMI.bEventAck; // Events Acknowledgement
	
//		(* Life bit *)
//			fbLifeBlink(tTimerValue:=T#500MS,bOut=>GV_CNC.stFanucData.stMagazineCNC.boLife); // Life bit Magazine->CNC
//			(*Fault*)
//			tonLifeON(IN:=GV_CNC.stFanucData.stCncMagazine.biLife,PT:=T#1000MS); // Life bit fault CNC->Magazine
//			tonLifeOFF(IN:=(NOT GV_CNC.stFanucData.stCncMagazine.biLife),PT:=T#1000MS); // Life bit fault CNC->Magazine
//			(*Reset Fault = Ack*)
//			IF GV_CNC.bEventAck THEN
//				GV_CNC.bAlLife:=FALSE;
//			END_IF
//			(*Set Fault*)
//			IF (tonLifeON.Q OR tonLifeOFF.Q) AND GV_CNC.bEnable=TRUE THEN
//				GV_CNC.bAlLife:=TRUE;
//			END_IF
//			(*Alarm 1 = Life bit*)	
//			IF GV_CNC.bAlLife THEN
//				GV_Events.aEventGroup[GV_CNC.iEventGroup].aAlarm[1].fbAlarm.ipArguments.Clear();
//				fbEventHMI(iEventGroup:=GV_CNC.iEventGroup,iIdEvent:=1,strEventType:='ALARM',bEventSet:=TRUE);
//			ELSE
//				fbEventHMI(iEventGroup:=GV_CNC.iEventGroup,iIdEvent:=1,strEventType:='ALARM',bEventSet:=FALSE);
//			END_IF
	
//		(* Alarm present *)
//		fbEventHMI.M_Event_Group_State(iEventGroup:=GV_CNC.iEventGroup,bEventPresence=>GV_Events.aEventGroup[GV_CNC.iEventGroup].bAlarmPresence);
	
//	(** OpMESSAGES **)
//		(* Message 1 = Nor ready *)
//			IF GV_Events.aEventGroup[GV_CNC.iEventGroup].bAlarmPresence=TRUE AND GV_CNC.bEnable=TRUE THEN
//				GV_Events.aEventGroup[GV_CNC.iEventGroup].aOpMessage[1].fbAlarm.ipArguments.Clear();
//				fbEventHMI(iEventGroup:=GV_CNC.iEventGroup,iIdEvent:=1,strEventType:='OpMESSAGE',bEventSet:=TRUE);
//			ELSE
//				fbEventHMI(iEventGroup:=GV_CNC.iEventGroup,iIdEvent:=1,strEventType:='OpMESSAGE',bEventSet:=FALSE);
//			END_IF

	
//	(** CNC MANAGEMENT **)
	
END_IF

END_FUNCTION_BLOCK

// ---- 12_Focas/03_POUs/01_PRGs/PRG_Focas.TcPOU
PROGRAM PRG_Focas
VAR
	(** INT **)
		iFocasLoop : INT := 0 ; // Use in a FOR Loop
		iLocationLoop : INT := 0 ; // Use in a FOR Loop
	
	(** FOCAS **)
		(** ARRAY **)
			aDataWrite : ARRAY [0..499] OF BYTE ;
			aDataRead : ARRAY [0..499] OF BYTE ;
			aData : ARRAY[1..256] OF BYTE ;
			aDataReset : ARRAY[1..256] OF BYTE ;
		
		(** STRING **)
		 sPartQuantity : STRING ;
		 
		(** DWORD **)
			dwTempDWORD : DWORD ;
			
		(** WORD **)
			wTempWORD : WORD ;
		
		(** REAL **)
			rTempParameter3 : REAL ;
			rTempParameter4 : REAL ;
			rTempParameter5 : REAL ;
			rTempREAL : REAL ;

		(** UINT **)
			uiAdrStartData : UINT ;
			uiAdrEndData : UINT ;
		
		(** INT **)
			iTempINT : INT ;
			iIndex : INT ;
			iDataIndex : INT ;
			
		(** BYTE **)
			byTempBYTE : BYTE ;
			byTypeData : BYTE ;
			byTypePMC : BYTE ;	
			byDataSize : BYTE ;
			byDataBitPos : BYTE ;
		
		(** FLAG **)
			bStartComm : BOOL ;
			bStartFocas : BOOL ;
			bStopFocas : BOOL ;
			bStart : BOOL ;
			bBarLenghtReaded : BOOL ;
		
		(** FB **)
			fb_ConnectionFocas : FB_ConnectionFocas ;
			fb_ReadFocas : FB_ReadFocas ;
			fb_WriteFocas : FB_WriteFocas ;
			tonWaitOpen : TON ;
END_VAR




			(* Update Tools in GV_Tool_Magazine *)
// 			FOR iFocasLoop:=1 TO GV_Tool_Magazine.iMaxAbsLocation BY 1 DO
// 				IF GV_Focas.stFocasMagazine.aToolParamIn[iFocasLoop].Location>0 THEN
// 					FOR iLocationLoop:=1 TO GV_Tool_Magazine.iMaxAbsLocation BY 1 DO
// 						IF GV_Tool_Magazine.aLocation[iLocationLoop].iRelLocationNumber=UINT_TO_INT(GV_Focas.stFocasMagazine.aToolParamIn[iFocasLoop].Location) THEN
// 							GV_Tool_Magazine.aLocation[iLocationLoop].stToolParam:=GV_Focas.stFocasMagazine.aToolParamIn[iFocasLoop]; // Tool Parameters
// 							GV_Tool_Magazine.aLocation[iLocationLoop].stToolName:=GV_Focas.stFocasMagazine.aToolNameIn[iFocasLoop]; // Tool Name
// 						END_IF
// 					END_FOR
// 				END_IF
// 			END_FOR

// 			GV_Focas.bWriteStart:=TRUE;
// 			GV_Focas.iWriteStep:=0;
// 			IF GV_Focas.bWriteStart AND GV_Focas.iWriteStep=0 AND (NOT fb_WriteFocas.bStartWrite) AND (NOT fb_WriteFocas.bBusy) THEN
// 				(* Copy Data in structure *)
// 				GV_Focas.iWriteStep:=1;
// 			END_IF
// 			IF GV_Focas.iWriteStep=1 THEN
// 				(* Parameter for Data *)
// 				GV_Focas.iWriteStep:=2;
// 			END_IF
// 			IF GV_Focas.iWriteStep=2 THEN
// 				(* End *)
// 					IF GV_CNC.Start_write_data_focas AND fb_WriteFocas.bDone THEN
// 						GV_Focas.iWriteStep:=0;
// 						GV_Focas.bWriteStart:=FALSE;
// 						GV_Focas.stFocasMagazine.bRefreshIn:=FALSE;
// 					END_IF
// 			END_IF

//-----------------------------------------------------------------------------------------
//
//                  					PRG_Focas
//
//								Gestion Echanges Focas		
//-----------------------------------------------------------------------------------------
//
//Auteur: G.GOETZ (inspired by S.MANTZER)
//Création: 19.02.2026
//Dernière modification : 19.02.2026 (G.GOETZ)
//       			
//-----------------------------------------------------------------------------------------
//
//     							Liste des modifications  	
//
// 19.02.2026 (G.GOETZ) -> Création		
//-----------------------------------------------------------------------------------------

//-----------------------------------------------------------------------------------------
// 									R5900-R5999 Available
//-----------------------------------------------------------------------------------------

(** Communication : Focas <-> Magazine **)
IF GV_CNC.bFocas THEN
			
	(* Start Focas *)
		IF GV_CNC.bEnable THEN
			bStartComm:=TRUE;
		ELSE
			bStartComm:=FALSE;
		END_IF
		
	(*Time to etablished Focas communication*)
		tonWaitOpen(IN:=bStartComm,PT:=T#30S);
		
	(*Call FB Communication Focas*)
		fb_ConnectionFocas(
							bStartComm:=tonWaitOpen.Q,
							bStopComm:=bStopFocas,
							iPortComm:=8193,
							SAdrCommFocas:=,
							sPathNameExe:='C:\WM\Soft\Focas\CommunicationADS-TC3.exe' ,
							sDirName:= 'C:\'
						  );
		
	(*Initialisation Reading and Writing data via Focas*)
		IF (NOT tonWaitOpen.Q) AND bStartComm THEN
			GV_CNC.bAlFocas:=TRUE; // Focas error
			(*For reading*)
				GV_CNC.stFanucData.stFocasData.bStartReadDataFocas:=FALSE;
				GV_CNC.stFanucData.stFocasData.iReadingPartDataStep:=0;
			(*For writing*)
				GV_CNC.stFanucData.stFocasData.bStartWriteDataFocas:=FALSE;		
				GV_CNC.stFanucData.stFocasData.iWritingPartDataStep:=0;
		END_IF
			
	(* Focas error *)
		IF GV_Focas.iReadErrorID<>0 OR GV_Focas.iWriteErrorID<>0 AND bStartComm THEN
			GV_CNC.bAlFocas:=TRUE;
			(*For reading*)
				GV_CNC.stFanucData.stFocasData.bStartReadDataFocas:=FALSE;
				GV_CNC.stFanucData.stFocasData.iReadingPartDataStep:=0;
			(*For writing*)
				GV_CNC.stFanucData.stFocasData.bStartWriteDataFocas:=FALSE;		
				GV_CNC.stFanucData.stFocasData.iWritingPartDataStep:=0;
			
			GV_Focas.bReadBusy:=FALSE;
			GV_Focas.bWriteBusy:=FALSE;
			GV_Focas.iReadErrorID:=0;
			GV_Focas.iWriteErrorID:=0;			
		END_IF

	(** Refresh Exchange IN : Focas -> Magazine **)
		GV_Focas.stFocasMagazine.bRefreshIn:=GV_General.bIsBlinking05s;
		IF GV_Focas.stFocasMagazine.bRefreshIn THEN
			GV_Focas.bReadStart:=TRUE;
 			GV_Focas.iReadStep:=0;
 			IF GV_Focas.bReadStart AND fb_ConnectionFocas.bFocasOk AND GV_Focas.iReadStep=0 AND GV_Focas.iWriteStep=0 AND (NOT fb_ReadFocas.bStartRead) AND (NOT fb_ReadFocas.bBusy) AND (NOT fb_ReadFocas.bDone) THEN
 				(* Copy Data in structure *)
					byTypePMC:=5;
					byTypeData:=0;
					uiAdrStartData:=5800;
					uiAdrEndData:=5800;
					byDataSize:=1;
 				GV_Focas.iWriteStep:=1;
 			END_IF
			IF GV_Focas.iReadStep=1 AND GV_Focas.bReadStart AND fb_ReadFocas.bDone THEN
 				GV_Focas.bReadStart:=FALSE;
				GV_Focas.iReadStep:=2;
			END_IF
			IF GV_Focas.iReadStep=2 THEN
 				//ICI;
				GV_Focas.stFocasMagazine.bRefreshIn:=FALSE;
			END_IF
		END_IF
	
	
	(** Refresh Exchange OUT : Magazine -> Focas **)
		GV_Focas.stMagazineFocas.bRefreshOut:=(NOT GV_General.bIsBlinking05s);
		IF GV_Focas.stMagazineFocas.bRefreshOut THEN
			GV_Focas.bWriteStart:=TRUE;
 			GV_Focas.iWriteStep:=0;
 			IF GV_Focas.bWriteStart AND fb_ConnectionFocas.bFocasOk AND GV_Focas.iReadStep=0 AND GV_Focas.iWriteStep=0 AND (NOT fb_WriteFocas.bStartWrite) AND (NOT fb_WriteFocas.bBusy) AND (NOT fb_WriteFocas.bDone) THEN
 				(* Copy Data in structure *)
					byTypePMC:=5;
					byTypeData:=0;
					uiAdrStartData:=5900;
					uiAdrEndData:=5900;
					byDataSize:=1;
 				GV_Focas.iWriteStep:=1;
 			END_IF
			IF GV_Focas.iWriteStep=1 AND GV_Focas.bWriteStart AND fb_WriteFocas.bDone THEN
 				GV_Focas.bWriteStart:=FALSE;
				GV_Focas.iWriteStep:=2;
			END_IF
			IF GV_Focas.iWriteStep=2 THEN
 				//ICI;
				GV_Focas.stMagazineFocas.bRefreshOut:=FALSE;
			END_IF
		END_IF
	
END_IF

END_PROGRAM

// ---- 12_Focas/03_POUs/02_FBs/FB_ConnectionFocas.TcPOU
FUNCTION_BLOCK FB_ConnectionFocas
VAR_INPUT
	(** STRING **)
		sPathNameExe : STRING ; // Chemin du fichier CommunicationADS-TC3.exe
		sDirName : STRING ; // Direction de l'emplacement de l'exécutable
		sAdrCommFocas : STRING ; // Adresse de la CNC pour établir la communication FOCAS
	
	(** INT **)
		iPortComm : INT ; // Port de communication
		
	(** FLAG **)	
		bStartComm : BOOL ; // Start de la communication FOCAS
		bStopComm : BOOL ; // Arrêt de la communication FOCAS
		bHidePrgGate : BOOL ; // Cacher le programme passerelle au démarrage
END_VAR
VAR_OUTPUT
	(** INT **)
		iErreurID : INT ; // Error ID
	
	(** FLAG **)
		bBusy : BOOL ; // Activer si le block fonction est en cours d'utilisation
		bDone : BOOL ; // Activer si le block fonction a correctement éxecuter
		bFocasAdsOk : BOOL ; // Commmunication ADS ok
		bFocasOk : BOOL ; // Communication Focas ok
END_VAR
VAR
	(** STRING **)
		sPathNameCmd : STRING := 'C:\Windows\System32\cmd.exe' ; // Chemin du fichier CommunicationADS-TC3.exe
		sCmdLine : STRING := 'C:\' ;
	
	(** BYTE **)
		bStep : BYTE := 0 ;
		bCptErrorOpenExe : BYTE := 0 ;
	
	(** FLAG **)
		bStartTimeOutOn	: BOOL ; // Start de la temporisation 
		bStartTimeOutOff : BOOL ; // Start de la temporisation 
	
	(** FB **)
		tonTimeOutAdsOn: TON ; // Temporisation pour vérifier la communication ADS
		tonTimeOutAdsOff : TON ; // Temporisation pour vérifier la communication ADS
		tonWaitNextOpen : TON ;
		ntStartCommAdsFocas	: NT_StartProcess ;
END_VAR

//-----------------------------------------------------------------------------------------
//
//                  			FB_ConnectionFocas
//
//								Connection Focas		
//-----------------------------------------------------------------------------------------
//
//Auteur: G.GOETZ (inspired by S.MANTZER)
//Création: 19.02.2026
//Dernière modification : 19.02.2026 (G.GOETZ)
//       			
//-----------------------------------------------------------------------------------------
//
//     							Liste des modifications  	
//
// 19.02.2026 (G.GOETZ) -> Création		
//-----------------------------------------------------------------------------------------

CASE bStep OF
	
	0:  // Ouverture automatique du programme passerelle
		IF bStartComm AND iErreurID=0 THEN
			// Build Command String
			sCmdLine:='/C '; // Special command indicating command string input
			sCmdLine:=CONCAT(sCmdLine,'start '); // Add start command
			sCmdLine:=CONCAT(sCmdLine,sPathNameExe); // Add target file
			bStep := 10;
		ELSE
			bBusy:=FALSE;
			bDone:=FALSE;
			sCmdLine:='';
		END_IF
		IF iErreurID<>0 AND (NOT bStartComm) THEN
			iErreurID:=0;
		END_IF
		IF bFocasAdsOk THEN
			bStep:=40;
		END_IF
	
	10:
		ntStartCommAdsFocas.START:=TRUE;
		IF ntStartCommAdsFocas.BUSY THEN
			bStep:=20;
		END_IF		
		IF ntStartCommAdsFocas.ERR THEN
			bStep:=100;
		END_IF
	
	20:
		IF (NOT ntStartCommAdsFocas.BUSY) THEN
			ntStartCommAdsFocas.START:=FALSE;
			bStep:=30;
		END_IF
		IF ntStartCommAdsFocas.ERR THEN
			bStep:=100;
		END_IF

	30:
		IF GV_Focas.bLifeFlag THEN
			bStep:=40;
		END_IF
		
		IF ntStartCommAdsFocas.ERR THEN
			bStep:=100;
		END_IF

	40:// Gestion de l'erreur lors de la communication ADS
		IF (NOT bFocasAdsOk) THEN
			bStep := 100;
		ELSIF bFocasAdsOk THEN
			iErreurID:=GV_Focas.iErrorAdsID;
		ELSE
			iErreurID:=0;
		END_IF
	
	100:
		tonWaitNextOpen.IN:=TRUE;
		IF tonWaitNextOpen.Q THEN
			tonWaitNextOpen.IN := FALSE;
			IF bCptErrorOpenExe<3 THEN
				bCptErrorOpenExe:=bCptErrorOpenExe+1;
				ntStartCommAdsFocas.START:=FALSE;
				bStep:=0;
			ELSE
				bCptErrorOpenExe:=0;
				
				iErreurID:=(-100);
				ntStartCommAdsFocas.START:=FALSE;
				bStep:=0;
			END_IF
		END_IF
		
END_CASE



// Mappage des variables 
	IF bFocasAdsOk THEN
		GV_Focas.iFocasPort:=iPortComm;
		GV_Focas.sFocasAdr:=sAdrCommFocas;
		GV_Focas.bFocasStartComm:=bStartComm;
		GV_Focas.bFocasStopComm:=bStopComm;
		GV_Focas.bFocasAdsOK:=bFocasAdsOk;
		
		bBusy:=GV_Focas.bFocasBusy;
		bDone:=GV_Focas.bFocasDone;
		bFocasOk:=GV_Focas.bFocasOk;
	ELSE
		GV_Focas.iFocasPort:=0;
		GV_Focas.sFocasAdr:='';
		GV_Focas.bFocasStartComm:=FALSE;
		GV_Focas.bFocasStopComm:=FALSE;
		GV_Focas.bFocasAdsOK:=FALSE;
		
		GV_Focas.bFocasBusy:=FALSE;
		GV_Focas.bFocasDone:=FALSE;
		GV_Focas.bFocasOk:=FALSE;
		
		bFocasOk:=FALSE;
	END_IF

A_LifeFlag();

ntStartCommAdsFocas(
	NETID:= '', 
	PATHSTR:= sPathNameCmd, 
	DIRNAME:= sDirName, 
	COMNDLINE:= sCmdLine, 
	START:= , 
	TMOUT:= , 
	BUSY=> , 
	ERR=> , 
	ERRID=> );
	
tonWaitNextOpen(IN:=,PT:=T#1S,Q=>,ET=>);

ACTION A_LifeFlag:
//-----------------------------------------------------------------------------------------
//
//                  				A_LifeFlag
//
//								Action Bit de Vie Focas		
//-----------------------------------------------------------------------------------------
//
//Auteur: G.GOETZ (inspired by S.MANTZER)
//Création: 19.02.2026
//Dernière modification : 19.02.2026 (G.GOETZ)
//       			
//-----------------------------------------------------------------------------------------
//
//     							Liste des modifications  	
//
// 19.02.2026 (G.GOETZ) -> Création		
//-----------------------------------------------------------------------------------------

IF GV_Focas.bLifeFlag THEN
	bStartTimeOutOn:=TRUE;
	bStartTimeOutOff:=FALSE;
	bFocasAdsOk:=TRUE;
END_IF

tonTimeOutAdsOn(IN := bStartTimeOutOn, pt := T#2S,);
IF tonTimeOutAdsOn.Q THEN
	bFocasAdsOk:=FALSE;
	GV_Focas.bFocasOK:=FALSE;
	bStartTimeOutOn:=FALSE;
	GV_Focas.bLifeFlag:=FALSE;
END_IF

IF bFocasAdsOk AND NOT GV_Focas.bLifeFlag THEN
	bStartTimeOutOff:=TRUE;
	bStartTimeOutOn:=FALSE;
END_IF

tonTimeOutAdsOff(IN := bStartTimeOutOff, pt := T#2S,);
IF tonTimeOutAdsOff.Q THEN
	bFocasAdsOk:=FALSE;
	bStartTimeOutOff:=FALSE;
END_IF
END_ACTION

END_FUNCTION_BLOCK

// ---- 12_Focas/03_POUs/02_FBs/FB_ReadFocas.TcPOU
FUNCTION_BLOCK FB_ReadFocas
VAR_INPUT
	(** UINT **)
		uiPMCAdr1 : UINT ; // Adresse de début de la donnée à lire
		uiPMCAdr2 : UINT ; // Adresse de fin de la donnée à lire
		uiGrandType : UINT ; // Grandeur du block de donnée à lire Exemple : data_type is 0(byte type) : length = 8 + N

	(** BYTE **)
		byTypePMC : BYTE ; // Type de variable à lire dans le PMC (G, R, X, Y...)
		byTypeData : BYTE ; // Type de donnée à lire (0 = byte, 1 = Word, 2 = Long, 3 = Bit, 4 = 32-bit floating-point type(30i-B Series/0i-F/PMi-A only), 5 = 64-bit floating-point type(30i-B Series/0i-F/PMi-A only)
	
	(** FLAG **)	
		bStartRead : BOOL := FALSE ;
		bBitRead : BYTE ; // Bit à lire dans le word du PMC
END_VAR
VAR_OUTPUT
	(** ARRAY **)
		aTabValLect : ARRAY [0..499] OF BYTE ; // Valeurs récupérées lors de la lecture		
		
	(** INT **)
		udiErrorID : INT ; // Error ID (0 == exécution ok)
		
	(** FLAG **)
		bBusy : BOOL := FALSE ; // Vrai si le bloc est en cours d'exécution
		bDone : BOOL := FALSE ; // Vrai si le bloc à terminé l'exécution sans erreur
		bError : BOOL := FALSE ; // Vrai si une erreur est survenue
END_VAR
VAR
	(** UINT **)
		uiTrueSizeRead : UINT ; // Table vérirable de la table à lire

	(** BYTE **)
		byIndexLect : BYTE := 0 ;

	(** FLAG **)	
		bErreurAff : BOOL := FALSE ; // Erreur lors de l'affectation, mauvaise valeur
		bTabEnvOk : BOOL := FALSE ;
END_VAR

//-----------------------------------------------------------------------------------------
//
//                  				FB_ReadFocas
//
//									Lecture Focas		
//-----------------------------------------------------------------------------------------
//
//Auteur: G.GOETZ (inspired by S.MANTZER)
//Création: 19.02.2026
//Dernière modification : 19.02.2026 (G.GOETZ)
//       			
//-----------------------------------------------------------------------------------------
//
//     							Liste des modifications  	
//
// 19.02.2026 (G.GOETZ) -> Création		
//-----------------------------------------------------------------------------------------

IF bStartRead AND (NOT GV_Focas.bReadDone) THEN
	
	IF byTypePMC>=0 AND byTypePMC<=13 THEN
		GV_Focas.stRead.uiTypePMC:=byTypePMC;
	ELSE
		bErreurAff := TRUE;
	END_IF
	
	IF byTypeData>=0 AND byTypeData<=5 THEN
		GV_Focas.stRead.uiTypeData:=byTypeData;
	ELSE
		bErreurAff := TRUE;
	END_IF
	
	IF (uiPMCAdr1>=0 AND uiPMCAdr1<=9499) AND (uiPMCAdr2>=0 AND uiPMCAdr2<=9499) THEN
		GV_Focas.stRead.uiPMCAdr1:=uiPMCAdr1;
		GV_Focas.stRead.uiPMCAdr2:=uiPMCAdr2;
		uiTrueSizeRead:=8+(uiPMCAdr2-uiPMCAdr1+1);
	ELSE
		bErreurAff := TRUE;		
	END_IF
	
	IF uiGrandType>=8 AND uiGrandType<=65535 THEN
		GV_Focas.stRead.uiGrandType:=uiGrandType;
	ELSE
		bErreurAff := TRUE;
	END_IF
	
	IF bBitRead>=0 AND bBitRead<=7 THEN
		GV_Focas.stRead.uiBitLect:=bBitRead;
	ELSE
		bErreurAff := TRUE;
	END_IF
	
	IF (NOT bErreurAff) THEN // Contrôle que le tableau soit remplis correctement et start de la lecture ou non
		GV_Focas.bReadStart:=TRUE;
		bTabEnvOk:=TRUE;
	ELSE
		GV_Focas.bReadStart:=FALSE;
		bError:=TRUE;
	END_IF
	
ELSE
	IF bTabEnvOk AND (NOT bStartRead) THEN // Réinitialisation du start après envoie et reset du start sur le bloc
		GV_Focas.bReadStart:=FALSE;
		bTabEnvOk:=FALSE;
	END_IF
	
	IF bError THEN // Réinitialisation des erreurs après le reset du start sur le bloc
		bError:=FALSE;
		bErreurAff:=FALSE;
	END_IF
END_IF

// Récupération des variables de sortie géré par le programme C#
	IF GV_Focas.bReadDone THEN
		aTabValLect:=GV_Focas.stRead.aTabValeur;
		udiErrorID:=GV_Focas.iReadErrorID;
	END_IF

// Test de la mise à jour du busy en temps réel
	bBusy:=GV_Focas.bReadBusy;
	bDone:=GV_Focas.bReadDone;

END_FUNCTION_BLOCK

// ---- 12_Focas/03_POUs/02_FBs/FB_WriteFocas.TcPOU
FUNCTION_BLOCK FB_WriteFocas
VAR_INPUT
	(** ARRAY **)	
		aTabEcriture : ARRAY [0..499] OF BYTE ; // Tableau des valeurs à écrire ([0] = première écriture, [1] = deuxième écriture)

	(** UINT **)
		uiPMCAdr1 : UINT ; // Adresse de début de la donnée à lire
		uiPMCAdr2 : UINT ; // Adresse de fin de la donnée à lire
		uiGrandType : UINT ; // Grandeur du block de donnée à lire Exemple : data_type is 0(byte type) : length = 8 + N
	
	(** BYTE **)			
		byBitWrite : BYTE ; // Valeur du bit pour l'écriture dans le PMC
		byTypePMC : BYTE ; // Type de variable à écrire dans le PMC
		byTypeData : BYTE ; // Type de donnée à lire (0 = byte, 1 = Word, 2 = Long, 4 = 32-bit floating-point type(30i-B Series/0i-F/PMi-A only), 5 = 64-bit floating-point type(30i-B Series/0i-F/PMi-A only)
		
	(** FLAG **)
		bStartWrite : BOOL ;
 
END_VAR
VAR_OUTPUT
	(** INT **)
		udiErrorID : INT ; // Error ID (0 == exécution ok)
		
	(** FLAG **)
		bBusy : BOOL := FALSE ; // Vrai si le bloc est en cours d'exécution
		bDone : BOOL := FALSE ; // Vrai si le bloc à terminé l'exécution sans erreur
		bError : BOOL := FALSE ; // Vrai si une erreur est survenue
END_VAR
VAR
	(** UINT **)
		uiGrandTypeBis : UINT ;
	
	(** INT **)
		iIndex : INT := 0 ; // Index
	
	(** FLAG **)
		bErreurAff : BOOL := FALSE ; // Erreur de saisie des différentes valeurs
		bErreurSaisi : BOOL := FALSE ;
END_VAR

//-----------------------------------------------------------------------------------------
//
//                  			FB_WriteFocas
//
//								Ecriture Focas		
//-----------------------------------------------------------------------------------------
//
//Auteur: G.GOETZ (inspired by S.MANTZER)
//Création: 19.02.2026
//Dernière modification : 19.02.2026 (G.GOETZ)
//       			
//-----------------------------------------------------------------------------------------
//
//     							Liste des modifications  	
//
// 19.02.2026 (G.GOETZ) -> Création		
//-----------------------------------------------------------------------------------------

IF bStartWrite AND (NOT GV_FOcas.bWriteDone) THEN	
		
	iIndex:=0; // Réinitialisation de l'index pour ajouter les valeurs au tableau
	FOR iIndex:=0 TO 499 BY 1 DO // Assignation des valeurs au tableau avec le contrôle des données saisies
		IF byTypeData=0 THEN // test de la saisie de la valeur en byte
			IF aTabEcriture[iIndex]>255 THEN
				bErreurSaisi:=TRUE;
			END_IF
		END_IF
		
		IF byTypeData=1 THEN // Test de la saisie de la valeur en Uint (Word)
			IF aTabEcriture[iIndex]>=0 AND aTabEcriture[iIndex]<=65535 THEN
				bErreurSaisi := TRUE;
			END_IF
		END_IF
		
		IF byTypeData=2 THEN // Test de la saisie de la valeur en Udint ( Long)
			IF aTabEcriture[iIndex]>=0 AND aTabEcriture[iIndex]<=4294967296 THEN
				bErreurSaisi:=TRUE;				
			END_IF
		END_IF
		
		IF byTypeData=3 THEN // Test de la saisie de la valeur en Bit (1 = true, 0 = false)
			IF aTabEcriture[iIndex]>=0 AND aTabEcriture[iIndex]<=1 THEN
				bErreurSaisi:=TRUE;
			END_IF
		END_IF
	END_FOR
	
	IF (NOT bErreurSaisi) THEN // Assigantion du tableau pour la récupération avec l'ADS
		GV_Focas.stWrite.aTabValeur:=aTabEcriture;
	END_IF
	
	IF byTypePMC>=0 AND byTypePMC<=13 THEN // Assignation des autres valeurs au tableau
		GV_Focas.stWrite.uiTypePMC:=byTypePMC;
	ELSE
		bErreurAff:=TRUE;
	END_IF
	
	IF byTypeData>=0 AND byTypeData<=5 THEN
		GV_Focas.stWrite.uiTypeData:=byTypeData;
	ELSE
		bErreurAff:=TRUE;
	END_IF
	
	IF (uiPMCAdr1>=0 AND uiPMCAdr1<=9499) AND (uiPMCAdr2>=0 AND uiPMCAdr2<=9499) THEN
		GV_Focas.stWrite.uiPMCAdr1:=uiPMCAdr1;
		GV_Focas.stWrite.uiPMCAdr2:=uiPMCAdr2;
	ELSE
		bErreurAff:=TRUE;		
	END_IF
	
	IF uiGrandType>=8 AND uiGrandType<=4010 THEN
		GV_Focas.stWrite.uiGrandType:=uiGrandType;
	ELSE
		bErreurAff:=TRUE;
	END_IF
	
	IF byBitWrite>=0 AND byBitWrite<=7 THEN
		GV_Focas.stWrite.uiBitLect:=byBitWrite;
	ELSE
		bErreurAff:=TRUE;
	END_IF
	
	IF (NOT bErreurAff) AND (NOT bErreurSaisi) THEN
		GV_Focas.bWriteStart:=TRUE;
	ELSE
		bError:=TRUE;
		bErreurAff:=FALSE;
		bErreurSaisi:=FALSE;
	END_IF
	
ELSE
	IF bError THEN
		GV_Focas.bWriteStart:=FALSE;
		bError:=FALSE;		
	END_IF
	
	IF (NOT bStartWrite) THEN // Réinitialisation du start après envoie et reset du start sur le bloc
		GV_Focas.bWriteStart:=FALSE;
	END_IF
END_IF

bBusy:=GV_Focas.bWriteBusy;
bDone:=GV_Focas.bWriteDone;
udiErrorID:=GV_Focas.iWriteErrorID;

END_FUNCTION_BLOCK

// ---- 13_HMI/03_POUs/01_PRGs/PRG_HMI.TcPOU
PROGRAM PRG_HMI
VAR
	(** R_TRIG **)	
		rtBlinkUp : R_TRIG ; 
		rtBlinkDown : R_TRIG ; 

	(** INT **)
		iAlarmLoop1 : INT ;
		iAlarmLoop2 : INT ;
		iMessageLoop1 : INT ; 
		iMessageLoop2 : INT ; 
END_VAR

//-----------------------------------------------------------------------------------------
//
//                  				PRG_HMI
//
//							Programme partie HMI    			
//-----------------------------------------------------------------------------------------
//
//Auteur: G.GOETZ
//Création: 28.01.2026
//Dernière modification : 28.01.2026 (G.GOETZ)
//       			
//-----------------------------------------------------------------------------------------
//
//     							Liste des modifications  	
//
// 28.01.2026 (G.GOETZ) -> Création	
//-----------------------------------------------------------------------------------------

(** PROCESS FLAG + R_Trig **)

	(* Button *)
		GV_HMI.rtEventAck(CLK:=GV_HMI.bButtonEventAck);
			GV_HMI.bEventAck:=GV_HMI.rtEventAck.Q;

		GV_HMI.rtINIT(CLK:=GV_HMI.bButtonInit);
		GV_HMI.rtAUTO(CLK:=GV_HMI.bButtonAUTO);
		GV_HMI.rtMANU(CLK:=GV_HMI.bButtonMANU);
		
		GV_HMI.stCycle.rtButtonStartStop(CLK:=GV_HMI.stCycle.bButtonStartStop);
		GV_HMI.stCycle.rtButtonStart(CLK:=GV_HMI.stCycle.bButtonStart);
		GV_HMI.stCycle.rtButtonStop(CLK:=GV_HMI.stCycle.bButtonStop);
		
		GV_HMI.rtReboot(CLK:=GV_HMI.bButtonReboot);
		GV_HMI.rtShutdown(CLK:=GV_HMI.bButtonShutdown);
		
		GV_HMI.rtHandwheelEnable(CLK:=GV_HMI.bButtonHandwheelEnable);
		GV_HMI.rtHandwheelIncr(CLK:=GV_HMI.bButtonHandwheelIncr);
		GV_HMI.rtHandwheelJog(CLK:=GV_HMI.bButtonHandwheelJog);
		
		//GV_HMI.rtRefreshToolMagazine(CLK:=GV_HMI.bButtonRefreshToolMagazine);
		GV_HMI.rtResetDataManipulator(CLK:=GV_HMI.bButtonResetDataManipulator);
		GV_HMI.rtResetDataChangingGripper1(CLK:=GV_HMI.bButtonResetDataChangingGripper1);
		GV_HMI.rtResetDataChangingGripper2(CLK:=GV_HMI.bButtonResetDataChangingGripper2);
		GV_HMI.rtResetDataSpindle(CLK:=GV_HMI.bButtonResetDataSpindle);

		GV_HMI.rtCncEnable(CLK:=GV_HMI.bButtonCncEnable);

		GV_HMI.stMagazineSettings.rtSettingsSave(CLK:=GV_HMI.stMagazineSettings.bButtonSettingsSave);
		
		GV_HMI.stManipulatorGripper.rtCloseManupulatorGripper(CLK:=GV_HMI.stManipulatorGripper.bButtonCloseManupulatorGripper);
		GV_HMI.stManipulatorGripper.rtOpenManupulatorGripper(CLK:=GV_HMI.stManipulatorGripper.bButtonOpenManupulatorGripper);

		GV_HMI.stCyltronic.rtButtonMoveRest(CLK:=GV_HMI.stCyltronic.bButtonMoveRest);
		GV_HMI.stCyltronic.rtButtonMoveWork(CLK:=GV_HMI.stCyltronic.bButtonMoveWork);
		
		GV_HMI.stAxes.rtButtonChoiceAxisX(CLK:=GV_HMI.stAxes.bButtonChoiceAxisX);
		GV_HMI.stAxes.rtButtonChoiceAxisY(CLK:=GV_HMI.stAxes.bButtonChoiceAxisY);
		GV_HMI.stAxes.rtButtonChoiceAxisZ(CLK:=GV_HMI.stAxes.bButtonChoiceAxisZ);
		GV_HMI.stAxes.rtButtonChoiceAxisArm(CLK:=GV_HMI.stAxes.bButtonChoiceAxisArm);
		GV_HMI.stAxes.rtButtonPlus(CLK:=GV_HMI.stAxes.bButtonPlus);
		GV_HMI.stAxes.rtButtonMinus(CLK:=GV_HMI.stAxes.bButtonMinus);

		GV_HMI.stAxes.rtButtonChoiceReferencingX(CLK:=GV_HMI.stAxes.bButtonChoiceReferencingX);
		GV_HMI.stAxes.rtButtonChoiceReferencingY(CLK:=GV_HMI.stAxes.bButtonChoiceReferencingY);
		GV_HMI.stAxes.rtButtonChoiceReferencingZ(CLK:=GV_HMI.stAxes.bButtonChoiceReferencingZ);
		GV_HMI.stAxes.rtButtonChoiceReferencingArm(CLK:=GV_HMI.stAxes.bButtonChoiceReferencingArm);
		GV_HMI.stAxes.rtButtonReferencingAxis(CLK:=GV_HMI.stAxes.bButtonReferencingAxis);
		
		GV_HMI.stAxes.rtButtonMinSofltLimit(CLK:=GV_HMI.stAxes.bButtonMinSofltLimit);
		GV_HMI.stAxes.rtButtonMaxSofltLimit(CLK:=GV_HMI.stAxes.bButtonMaxSofltLimit);
		
		GV_HMI.stMagazineTeach.rtTeachLocation(CLK:=GV_HMI.stMagazineTeach.bButtonTeachLocation);
		GV_HMI.stMagazineTeach.rtTeachRack(CLK:=GV_HMI.stMagazineTeach.bButtonTeachRack);
		GV_HMI.stMagazineTeach.rtTeachAllTop(CLK:=GV_HMI.stMagazineTeach.bButtonTeachAllTop);
		GV_HMI.stMagazineTeach.rtTeachAllBottom(CLK:=GV_HMI.stMagazineTeach.bButtonTeachAllBottom);

		GV_HMI.stBackup.rtButtonProject(CLK:=GV_HMI.stBackup.bButtonProject);
		GV_HMI.stBackup.rtButtonInitData(CLK:=GV_HMI.stBackup.bButtonInitData);
		GV_HMI.stBackup.rtButtonExportData(CLK:=GV_HMI.stBackup.bButtonExportData);
		GV_HMI.stBackup.rtButtonImportData(CLK:=GV_HMI.stBackup.bButtonImportData);
		
		GV_HMI.stBackup.rtButtonExportAlarms(CLK:=GV_HMI.stBackup.bButtonExportAlarms);
		GV_HMI.stBackup.rtButtonExportMessages(CLK:=GV_HMI.stBackup.bButtonExportMessages);
		
